(* Logix 5000 project; controller reports 1756-L63 rev 20.15; software revision 20.04; part 36 of 52 *)

        [42].log_data[40].minminute := 21, [42].log_data[40].maxminute := 25, [42].log_data[40].valid := 1, [42].log_data[41].min := 0.03412134, [42].log_data[41].max := 0.04962842, [42].log_data[41].total := 152.0447, [42].log_data[41].time := 3600.0, [42].log_data[41].minminute := 8, [42].log_data[41].maxminute := 47, [42].log_data[41].valid := 1, [42].log_data[42].min := 2.2923493, [42].log_data[42].max := 2.2970603, [42].log_data[42].total := 8261.717, [42].log_data[42].time := 3600.0, [42].log_data[42].minminute := 49, [42].log_data[42].maxminute := 24, [42].log_data[42].valid := 1, [42].log_data[43].min := -0.27999878, [42].log_data[43].max := -0.26000214, [42].log_data[43].total := -1007.5765, [42].log_data[43].time := 3600.0, [42].log_data[43].valid := 1, [42].log_data[44].min := -0.3199997, [42].log_data[44].max := -0.30000305, [42].log_data[44].total := -1084.2107, [42].log_data[44].time := 3600.0, [42].log_data[44].minminute := 1, [42].log_data[44].valid := 1, [42].log_data[45].time := 3600.0, [42].log_data[45].valid := 1, [42].log_data[46].time := 3600.0, [42].log_data[46].valid := 1, [42].log_data[47].time := 3600.0, [42].log_data[47].valid := 1, [42].log_data[48].min := 6.5827026, [42].log_data[48].max := 6.9506707, [42].log_data[48].total := 24231.43, [42].log_data[48].time := 3600.0, [42].log_data[48].minminute := 26, [42].log_data[48].maxminute := 3, [42].log_data[48].valid := 1, [42].log_data[49].min := 7.0381904, [42].log_data[49].max := 9.47083, [42].log_data[49].total := 29556.547, [42].log_data[49].time := 3600.0, [42].log_data[49].minminute := 23, [42].log_data[49].maxminute := 59, [42].log_data[49].valid := 1, [42].log_data[50].min := 2.0538552, [42].log_data[50].max := 2.1284068, [42].log_data[50].total := 7533.663, [42].log_data[50].time := 3600.0, [42].log_data[50].minminute := 59, [42].log_data[50].maxminute := 6, [42].log_data[50].valid := 1, [42].log_data[51].time := 3600.0, [42].log_data[51].valid := 1, [42].log_data[52].min := -2.959999, [42].log_data[52].max := 0.11999512, [42].log_data[52].total := -7758.8574,
        [42].log_data[52].time := 3600.0, [42].log_data[52].valid := 1, [42].log_data[53].min := -2.7400055, [42].log_data[53].max := 0.27999878, [42].log_data[53].total := -7175.7085, [42].log_data[53].time := 3600.0, [42].log_data[53].minminute := 37, [42].log_data[53].maxminute := 5, [42].log_data[53].valid := 1, [42].log_data[54].max := 0.538, [42].log_data[54].total := 1231.8954, [42].log_data[54].time := 3600.0, [42].log_data[54].maxminute := 11, [42].log_data[54].valid := 1, [42].log_data[55].max := 0.568, [42].log_data[55].total := 1217.1237, [42].log_data[55].time := 3600.0, [42].log_data[55].minminute := 4, [42].log_data[55].maxminute := 37, [42].log_data[55].valid := 1, [42].log_data[56].min := 0.16024561, [42].log_data[56].max := 0.1607167, [42].log_data[56].total := 577.47437, [42].log_data[56].time := 3600.0, [42].log_data[56].minminute := 10, [42].log_data[56].maxminute := 50, [42].log_data[56].valid := 1, [42].log_data[57].min := 0.28492987, [42].log_data[57].max := 0.28661802, [42].log_data[57].total := 1028.5197, [42].log_data[57].time := 3600.0, [42].log_data[57].minminute := 47, [42].log_data[57].maxminute := 1, [42].log_data[57].valid := 1, [42].log_data[58].time := 3600.0, [42].log_data[58].valid := 1, [42].log_data[59].time := 3600.0, [42].log_data[59].valid := 1, [42].log_data[60].valid := 1, [42].log_data[61].valid := 1, [42].log_data[62].valid := 1, [42].log_data[63].valid := 1, [42].log_data[64].valid := 1, [42].log_data[65].valid := 1, [42].log_data[66].valid := 1, [42].log_data[67].valid := 1, [42].log_data[68].valid := 1, [42].log_data[69].valid := 1, [42].log_data[70].valid := 1, [42].log_data[71].valid := 1, [42].log_data[72].valid := 1, [42].log_data[73].valid := 1, [42].log_data[74].valid := 1, [42].log_data[75].valid := 1, [42].log_data[76].valid := 1, [42].log_data[77].valid := 1, [42].log_data[78].valid := 1, [42].log_data[79].valid := 1, [42].log_data[80].valid := 1, [42].log_data[81].valid := 1,
        [42].log_data[82].valid := 1, [42].log_data[83].valid := 1, [42].log_data[84].valid := 1, [42].log_data[85].valid := 1, [42].log_data[86].valid := 1, [42].log_data[87].valid := 1, [42].log_data[88].valid := 1, [42].log_data[89].valid := 1, [42].log_data[90].valid := 1, [42].log_data[91].valid := 1, [42].log_data[92].valid := 1, [42].log_data[93].valid := 1, [42].log_data[94].valid := 1, [42].log_data[95].valid := 1, [42].log_data[96].valid := 1, [42].log_data[97].valid := 1, [42].log_data[98].valid := 1, [42].log_data[99].valid := 1, [42].log_data[100].valid := 1, [42].log_data[101].valid := 1, [42].log_data[102].valid := 1, [42].log_data[103].valid := 1, [42].log_data[104].valid := 1, [42].log_data[105].valid := 1, [42].log_data[106].valid := 1, [42].log_data[107].valid := 1, [42].log_data[108].valid := 1, [42].log_data[109].valid := 1, [42].log_data[110].valid := 1, [42].log_data[111].valid := 1, [42].log_data[112].valid := 1, [42].log_data[113].valid := 1, [42].log_data[114].valid := 1, [42].log_data[115].valid := 1, [42].log_data[116].valid := 1, [42].log_data[117].valid := 1, [42].log_data[118].valid := 1, [42].log_data[119].valid := 1, [42].log_data[120].valid := 1, [42].log_data[121].valid := 1, [42].log_data[122].valid := 1, [42].log_data[123].valid := 1, [42].log_data[124].valid := 1, [42].time.Year := 2023, [42].time.Month := 1, [42].time.Day := 14, [42].time.Hour := 21, [42].time.Minute := 59, [42].time.Second := 59, [43].log_data[0].min := 1.0, [43].log_data[0].max := 1.0, [43].log_data[0].total := 3600.0, [43].log_data[0].time := 3600.0, [43].log_data[0].valid := 1, [43].log_data[1].max := 1.0, [43].log_data[1].total := 564.5, [43].log_data[1].time := 3600.0, [43].log_data[1].maxminute := 21, [43].log_data[1].valid := 1, [43].log_data[2].max := 1.0,
        [43].log_data[2].total := 561.0, [43].log_data[2].time := 3600.0, [43].log_data[2].maxminute := 21, [43].log_data[2].valid := 1, [43].log_data[3].time := 3600.0, [43].log_data[3].valid := 1, [43].log_data[4].time := 3600.0, [43].log_data[4].valid := 1, [43].log_data[5].max := 1.0, [43].log_data[5].total := 239.5, [43].log_data[5].time := 3600.0, [43].log_data[5].maxminute := 22, [43].log_data[5].valid := 1, [43].log_data[6].time := 3600.0, [43].log_data[6].valid := 1, [43].log_data[7].time := 3600.0, [43].log_data[7].valid := 1, [43].log_data[8].min := 1.0, [43].log_data[8].max := 1.0, [43].log_data[8].total := 3600.0, [43].log_data[8].time := 3600.0, [43].log_data[8].valid := 1, [43].log_data[9].min := 1.0, [43].log_data[9].max := 1.0, [43].log_data[9].total := 3600.0, [43].log_data[9].time := 3600.0, [43].log_data[9].valid := 1, [43].log_data[10].min := 1.0, [43].log_data[10].max := 1.0, [43].log_data[10].total := 3600.0, [43].log_data[10].time := 3600.0, [43].log_data[10].valid := 1, [43].log_data[11].time := 3600.0, [43].log_data[11].valid := 1, [43].log_data[12].min := 1.0, [43].log_data[12].max := 1.0, [43].log_data[12].total := 3600.0, [43].log_data[12].time := 3600.0, [43].log_data[12].valid := 1, [43].log_data[13].min := 1.0, [43].log_data[13].max := 1.0, [43].log_data[13].total := 3600.0, [43].log_data[13].time := 3600.0, [43].log_data[13].valid := 1, [43].log_data[14].time := 3600.0, [43].log_data[14].valid := 1, [43].log_data[15].time := 3600.0, [43].log_data[15].valid := 1, [43].log_data[16].time := 3600.0, [43].log_data[16].valid := 1, [43].log_data[17].min := 1.0, [43].log_data[17].max := 1.0, [43].log_data[17].total := 3600.0, [43].log_data[17].time := 3600.0, [43].log_data[17].valid := 1, [43].log_data[18].time := 3600.0, [43].log_data[18].valid := 1, [43].log_data[19].time := 3600.0, [43].log_data[19].valid := 1, [43].log_data[20].time := 3600.0,
        [43].log_data[20].valid := 1, [43].log_data[21].min := 1.0, [43].log_data[21].max := 1.0, [43].log_data[21].total := 3600.0, [43].log_data[21].time := 3600.0, [43].log_data[21].valid := 1, [43].log_data[22].time := 3600.0, [43].log_data[22].valid := 1, [43].log_data[23].time := 3600.0, [43].log_data[23].valid := 1, [43].log_data[24].time := 3600.0, [43].log_data[24].valid := 1, [43].log_data[25].time := 3600.0, [43].log_data[25].valid := 1, [43].log_data[26].time := 3600.0, [43].log_data[26].valid := 1, [43].log_data[27].time := 3600.0, [43].log_data[27].valid := 1, [43].log_data[28].time := 3600.0, [43].log_data[28].valid := 1, [43].log_data[29].min := 1.0, [43].log_data[29].max := 1.0, [43].log_data[29].total := 3600.0, [43].log_data[29].time := 3600.0, [43].log_data[29].valid := 1, [43].log_data[30].min := 1.0, [43].log_data[30].max := 1.0, [43].log_data[30].total := 3600.0, [43].log_data[30].time := 3600.0, [43].log_data[30].valid := 1, [43].log_data[31].max := 1.0, [43].log_data[31].total := 1629.998, [43].log_data[31].time := 3600.0, [43].log_data[31].maxminute := 3, [43].log_data[31].valid := 1, [43].log_data[32].max := 1.0, [43].log_data[32].total := 1440.998, [43].log_data[32].time := 3600.0, [43].log_data[32].minminute := 2, [43].log_data[32].valid := 1, [43].log_data[33].time := 3600.0, [43].log_data[33].valid := 1, [43].log_data[34].time := 3600.0, [43].log_data[34].valid := 1, [43].log_data[35].max := 1.0, [43].log_data[35].total := 1536.498, [43].log_data[35].time := 3600.0, [43].log_data[35].minminute := 7, [43].log_data[35].valid := 1, [43].log_data[36].max := 1.0, [43].log_data[36].total := 1622.2471, [43].log_data[36].time := 3600.0, [43].log_data[36].maxminute := 8, [43].log_data[36].valid := 1, [43].log_data[37].max := 7.23916, [43].log_data[37].total := 3552.5513, [43].log_data[37].time := 3600.0, [43].log_data[37].maxminute := 23, [43].log_data[37].valid := 1, [43].log_data[38].time := 3600.0,
        [43].log_data[38].valid := 1, [43].log_data[39].min := 0.997415, [43].log_data[39].max := 1.0214411, [43].log_data[39].total := 3638.9631, [43].log_data[39].time := 3600.0, [43].log_data[39].minminute := 29, [43].log_data[39].maxminute := 26, [43].log_data[39].valid := 1, [43].log_data[40].min := 7.5816298, [43].log_data[40].max := 7.5865765, [43].log_data[40].total := 27307.055, [43].log_data[40].time := 3600.0, [43].log_data[40].minminute := 41, [43].log_data[40].maxminute := 2, [43].log_data[40].valid := 1, [43].log_data[41].min := 0.03785083, [43].log_data[41].max := 0.056694824, [43].log_data[41].total := 165.39845, [43].log_data[41].time := 3600.0, [43].log_data[41].minminute := 46, [43].log_data[41].maxminute := 20, [43].log_data[41].valid := 1, [43].log_data[42].min := 2.2922316, [43].log_data[42].max := 2.2970603, [43].log_data[42].total := 8261.55, [43].log_data[42].time := 3600.0, [43].log_data[42].minminute := 23, [43].log_data[42].maxminute := 1, [43].log_data[42].valid := 1, [43].log_data[43].min := -0.27999878, [43].log_data[43].max := -0.26000214, [43].log_data[43].total := -1007.7663, [43].log_data[43].time := 3600.0, [43].log_data[43].maxminute := 10, [43].log_data[43].valid := 1, [43].log_data[44].min := -0.3199997, [43].log_data[44].max := -0.30000305, [43].log_data[44].total := -1084.6222, [43].log_data[44].time := 3600.0, [43].log_data[44].valid := 1, [43].log_data[45].time := 3600.0, [43].log_data[45].valid := 1, [43].log_data[46].time := 3600.0, [43].log_data[46].valid := 1, [43].log_data[47].time := 3600.0, [43].log_data[47].valid := 1, [43].log_data[48].min := 6.5794053, [43].log_data[48].max := 6.9666095, [43].log_data[48].total := 24206.664, [43].log_data[48].time := 3600.0, [43].log_data[48].minminute := 53, [43].log_data[48].maxminute := 29, [43].log_data[48].valid := 1, [43].log_data[49].min := 6.964974, [43].log_data[49].max := 9.644745, [43].log_data[49].total := 30286.188, [43].log_data[49].time := 3600.0, [43].log_data[49].minminute := 49, [43].log_data[49].maxminute := 20, [43].log_data[49].valid := 1,
        [43].log_data[50].min := 2.0134585, [43].log_data[50].max := 2.1326468, [43].log_data[50].total := 7487.468, [43].log_data[50].time := 3600.0, [43].log_data[50].minminute := 22, [43].log_data[50].maxminute := 30, [43].log_data[50].valid := 1, [43].log_data[51].time := 3600.0, [43].log_data[51].valid := 1, [43].log_data[52].min := -2.959999, [43].log_data[52].max := 0.11999512, [43].log_data[52].total := -7728.6436, [43].log_data[52].time := 3600.0, [43].log_data[52].minminute := 4, [43].log_data[52].maxminute := 2, [43].log_data[52].valid := 1, [43].log_data[53].min := -2.5200043, [43].log_data[53].max := 0.27999878, [43].log_data[53].total := -7386.8955, [43].log_data[53].time := 3600.0, [43].log_data[53].minminute := 55, [43].log_data[53].maxminute := 51, [43].log_data[53].valid := 1, [43].log_data[54].max := 0.523, [43].log_data[54].total := 1217.3251, [43].log_data[54].time := 3600.0, [43].log_data[54].minminute := 2, [43].log_data[54].maxminute := 25, [43].log_data[54].valid := 1, [43].log_data[55].max := 0.522, [43].log_data[55].total := 1254.3055, [43].log_data[55].time := 3600.0, [43].log_data[55].minminute := 7, [43].log_data[55].maxminute := 40, [43].log_data[55].valid := 1, [43].log_data[56].min := 0.16020635, [43].log_data[56].max := 0.16067745, [43].log_data[56].total := 577.47656, [43].log_data[56].time := 3600.0, [43].log_data[56].minminute := 57, [43].log_data[56].maxminute := 11, [43].log_data[56].valid := 1, [43].log_data[57].min := 0.28355587, [43].log_data[57].max := 0.28532246, [43].log_data[57].total := 1025.724, [43].log_data[57].time := 3600.0, [43].log_data[57].minminute := 59, [43].log_data[57].maxminute := 11, [43].log_data[57].valid := 1, [43].log_data[58].time := 3600.0, [43].log_data[58].valid := 1, [43].log_data[59].time := 3600.0, [43].log_data[59].valid := 1, [43].log_data[60].valid := 1, [43].log_data[61].valid := 1, [43].log_data[62].valid := 1, [43].log_data[63].valid := 1, [43].log_data[64].valid := 1, [43].log_data[65].valid := 1, [43].log_data[66].valid := 1,
        [43].log_data[67].valid := 1, [43].log_data[68].valid := 1, [43].log_data[69].valid := 1, [43].log_data[70].valid := 1, [43].log_data[71].valid := 1, [43].log_data[72].valid := 1, [43].log_data[73].valid := 1, [43].log_data[74].valid := 1, [43].log_data[75].valid := 1, [43].log_data[76].valid := 1, [43].log_data[77].valid := 1, [43].log_data[78].valid := 1, [43].log_data[79].valid := 1, [43].log_data[80].valid := 1, [43].log_data[81].valid := 1, [43].log_data[82].valid := 1, [43].log_data[83].valid := 1, [43].log_data[84].valid := 1, [43].log_data[85].valid := 1, [43].log_data[86].valid := 1, [43].log_data[87].valid := 1, [43].log_data[88].valid := 1, [43].log_data[89].valid := 1, [43].log_data[90].valid := 1, [43].log_data[91].valid := 1, [43].log_data[92].valid := 1, [43].log_data[93].valid := 1, [43].log_data[94].valid := 1, [43].log_data[95].valid := 1, [43].log_data[96].valid := 1, [43].log_data[97].valid := 1, [43].log_data[98].valid := 1, [43].log_data[99].valid := 1, [43].log_data[100].valid := 1, [43].log_data[101].valid := 1, [43].log_data[102].valid := 1, [43].log_data[103].valid := 1, [43].log_data[104].valid := 1, [43].log_data[105].valid := 1, [43].log_data[106].valid := 1, [43].log_data[107].valid := 1, [43].log_data[108].valid := 1, [43].log_data[109].valid := 1, [43].log_data[110].valid := 1, [43].log_data[111].valid := 1, [43].log_data[112].valid := 1, [43].log_data[113].valid := 1, [43].log_data[114].valid := 1, [43].log_data[115].valid := 1, [43].log_data[116].valid := 1, [43].log_data[117].valid := 1, [43].log_data[118].valid := 1, [43].log_data[119].valid := 1, [43].log_data[120].valid := 1, [43].log_data[121].valid := 1, [43].log_data[122].valid := 1, [43].log_data[123].valid := 1, [43].log_data[124].valid := 1, [43].time.Year := 2023, [43].time.Month := 1,
        [43].time.Day := 14, [43].time.Hour := 22, [43].time.Minute := 59, [43].time.Second := 59, [44].log_data[0].min := 1.0, [44].log_data[0].max := 1.0, [44].log_data[0].total := 3599.5, [44].log_data[0].time := 3599.5, [44].log_data[0].valid := 1, [44].log_data[1].max := 1.0, [44].log_data[1].total := 535.5, [44].log_data[1].time := 3599.5, [44].log_data[1].maxminute := 50, [44].log_data[1].valid := 1, [44].log_data[2].max := 1.0, [44].log_data[2].total := 532.0, [44].log_data[2].time := 3599.5, [44].log_data[2].maxminute := 50, [44].log_data[2].valid := 1, [44].log_data[3].time := 3599.5, [44].log_data[3].valid := 1, [44].log_data[4].time := 3599.5, [44].log_data[4].valid := 1, [44].log_data[5].max := 1.0, [44].log_data[5].total := 227.5, [44].log_data[5].time := 3599.5, [44].log_data[5].maxminute := 51, [44].log_data[5].valid := 1, [44].log_data[6].time := 3599.5, [44].log_data[6].valid := 1, [44].log_data[7].time := 3599.5, [44].log_data[7].valid := 1, [44].log_data[8].min := 1.0, [44].log_data[8].max := 1.0, [44].log_data[8].total := 3599.5, [44].log_data[8].time := 3599.5, [44].log_data[8].valid := 1, [44].log_data[9].min := 1.0, [44].log_data[9].max := 1.0, [44].log_data[9].total := 3599.5, [44].log_data[9].time := 3599.5, [44].log_data[9].valid := 1, [44].log_data[10].min := 1.0, [44].log_data[10].max := 1.0, [44].log_data[10].total := 3599.5, [44].log_data[10].time := 3599.5, [44].log_data[10].valid := 1, [44].log_data[11].time := 3599.5, [44].log_data[11].valid := 1, [44].log_data[12].min := 1.0, [44].log_data[12].max := 1.0, [44].log_data[12].total := 3599.5, [44].log_data[12].time := 3599.5, [44].log_data[12].valid := 1, [44].log_data[13].min := 1.0, [44].log_data[13].max := 1.0, [44].log_data[13].total := 3599.5, [44].log_data[13].time := 3599.5, [44].log_data[13].valid := 1, [44].log_data[14].time := 3599.5,
        [44].log_data[14].valid := 1, [44].log_data[15].time := 3599.5, [44].log_data[15].valid := 1, [44].log_data[16].time := 3599.5, [44].log_data[16].valid := 1, [44].log_data[17].min := 1.0, [44].log_data[17].max := 1.0, [44].log_data[17].total := 3599.5, [44].log_data[17].time := 3599.5, [44].log_data[17].valid := 1, [44].log_data[18].time := 3599.5, [44].log_data[18].valid := 1, [44].log_data[19].time := 3599.5, [44].log_data[19].valid := 1, [44].log_data[20].time := 3599.5, [44].log_data[20].valid := 1, [44].log_data[21].min := 1.0, [44].log_data[21].max := 1.0, [44].log_data[21].total := 3599.5, [44].log_data[21].time := 3599.5, [44].log_data[21].valid := 1, [44].log_data[22].time := 3599.5, [44].log_data[22].valid := 1, [44].log_data[23].time := 3599.5, [44].log_data[23].valid := 1, [44].log_data[24].time := 3599.5, [44].log_data[24].valid := 1, [44].log_data[25].time := 3599.5, [44].log_data[25].valid := 1, [44].log_data[26].time := 3599.5, [44].log_data[26].valid := 1, [44].log_data[27].time := 3599.5, [44].log_data[27].valid := 1, [44].log_data[28].time := 3599.5, [44].log_data[28].valid := 1, [44].log_data[29].min := 1.0, [44].log_data[29].max := 1.0, [44].log_data[29].total := 3599.5, [44].log_data[29].time := 3599.5, [44].log_data[29].valid := 1, [44].log_data[30].min := 1.0, [44].log_data[30].max := 1.0, [44].log_data[30].total := 3599.5, [44].log_data[30].time := 3599.5, [44].log_data[30].valid := 1, [44].log_data[31].max := 1.0, [44].log_data[31].total := 1629.7471, [44].log_data[31].time := 3599.5, [44].log_data[31].maxminute := 7, [44].log_data[31].valid := 1, [44].log_data[32].max := 1.0, [44].log_data[32].total := 1440.498, [44].log_data[32].time := 3599.5, [44].log_data[32].minminute := 5, [44].log_data[32].valid := 1, [44].log_data[33].time := 3599.5, [44].log_data[33].valid := 1, [44].log_data[34].time := 3599.5, [44].log_data[34].valid := 1, [44].log_data[35].max := 1.0,
        [44].log_data[35].total := 1629.7471, [44].log_data[35].time := 3599.5, [44].log_data[35].maxminute := 1, [44].log_data[35].valid := 1, [44].log_data[36].max := 1.0, [44].log_data[36].total := 1440.2471, [44].log_data[36].time := 3599.5, [44].log_data[36].valid := 1, [44].log_data[37].max := 7.5873804, [44].log_data[37].total := 3523.6545, [44].log_data[37].time := 3599.5, [44].log_data[37].maxminute := 52, [44].log_data[37].valid := 1, [44].log_data[38].time := 3599.5, [44].log_data[38].valid := 1, [44].log_data[39].min := 0.99859273, [44].log_data[39].max := 1.0223833, [44].log_data[39].total := 3639.1343, [44].log_data[39].time := 3599.5, [44].log_data[39].minminute := 53, [44].log_data[39].maxminute := 51, [44].log_data[39].valid := 1, [44].log_data[40].min := 7.5703626, [44].log_data[40].max := 7.592072, [44].log_data[40].total := 27304.006, [44].log_data[40].time := 3599.5, [44].log_data[40].minminute := 57, [44].log_data[40].maxminute := 58, [44].log_data[40].valid := 1, [44].log_data[41].min := 0.029802978, [44].log_data[41].max := 0.044524662, [44].log_data[41].total := 127.272896, [44].log_data[41].time := 3599.5, [44].log_data[41].minminute := 15, [44].log_data[41].valid := 1, [44].log_data[42].min := 2.2921138, [44].log_data[42].max := 2.2970603, [44].log_data[42].total := 8260.388, [44].log_data[42].time := 3599.5, [44].log_data[42].minminute := 50, [44].log_data[42].maxminute := 11, [44].log_data[42].valid := 1, [44].log_data[43].min := -0.27999878, [44].log_data[43].max := -0.26000214, [44].log_data[43].total := -1004.873, [44].log_data[43].time := 3599.5, [44].log_data[43].valid := 1, [44].log_data[44].min := -0.3199997, [44].log_data[44].max := -0.30000305, [44].log_data[44].total := -1081.1991, [44].log_data[44].time := 3599.5, [44].log_data[44].valid := 1, [44].log_data[45].time := 3599.5, [44].log_data[45].valid := 1, [44].log_data[46].time := 3599.5, [44].log_data[46].valid := 1, [44].log_data[47].time := 3599.5, [44].log_data[47].valid := 1, [44].log_data[48].min := 6.690153, [44].log_data[48].max := 6.9295106,
        [44].log_data[48].total := 24392.291, [44].log_data[48].time := 3599.5, [44].log_data[48].maxminute := 57, [44].log_data[48].valid := 1, [44].log_data[49].min := 7.833956, [44].log_data[49].max := 9.64494, [44].log_data[49].total := 33088.74, [44].log_data[49].time := 3599.5, [44].log_data[49].maxminute := 50, [44].log_data[49].valid := 1, [44].log_data[50].min := 2.006392, [44].log_data[50].max := 2.1253445, [44].log_data[50].total := 7408.252, [44].log_data[50].time := 3599.5, [44].log_data[50].minminute := 51, [44].log_data[50].maxminute := 57, [44].log_data[50].valid := 1, [44].log_data[51].time := 3599.5, [44].log_data[51].valid := 1, [44].log_data[52].min := -3.0999985, [44].log_data[52].max := 0.11999512, [44].log_data[52].total := -7716.6855, [44].log_data[52].time := 3599.5, [44].log_data[52].minminute := 7, [44].log_data[52].maxminute := 5, [44].log_data[52].valid := 1, [44].log_data[53].min := -2.5, [44].log_data[53].max := 0.27999878, [44].log_data[53].total := -7181.388, [44].log_data[53].time := 3599.5, [44].log_data[53].minminute := 4, [44].log_data[53].maxminute := 43, [44].log_data[53].valid := 1, [44].log_data[54].max := 0.55149996, [44].log_data[54].total := 1217.8906, [44].log_data[54].time := 3599.5, [44].log_data[54].minminute := 5, [44].log_data[54].maxminute := 49, [44].log_data[54].valid := 1, [44].log_data[55].max := 0.5395, [44].log_data[55].total := 1217.0914, [44].log_data[55].time := 3599.5, [44].log_data[55].maxminute := 22, [44].log_data[55].valid := 1, [44].log_data[56].min := 0.16028486, [44].log_data[56].max := 0.16063818, [44].log_data[56].total := 577.4504, [44].log_data[56].time := 3599.5, [44].log_data[56].minminute := 14, [44].log_data[56].maxminute := 3, [44].log_data[56].valid := 1, [44].log_data[57].min := 0.2833203, [44].log_data[57].max := 0.2837129, [44].log_data[57].total := 1020.4592, [44].log_data[57].time := 3599.5, [44].log_data[57].minminute := 32, [44].log_data[57].valid := 1, [44].log_data[58].time := 3599.5, [44].log_data[58].valid := 1, [44].log_data[59].time := 3599.5,
        [44].log_data[59].valid := 1, [44].log_data[60].valid := 1, [44].log_data[61].valid := 1, [44].log_data[62].valid := 1, [44].log_data[63].valid := 1, [44].log_data[64].valid := 1, [44].log_data[65].valid := 1, [44].log_data[66].valid := 1, [44].log_data[67].valid := 1, [44].log_data[68].valid := 1, [44].log_data[69].valid := 1, [44].log_data[70].valid := 1, [44].log_data[71].valid := 1, [44].log_data[72].valid := 1, [44].log_data[73].valid := 1, [44].log_data[74].valid := 1, [44].log_data[75].valid := 1, [44].log_data[76].valid := 1, [44].log_data[77].valid := 1, [44].log_data[78].valid := 1, [44].log_data[79].valid := 1, [44].log_data[80].valid := 1, [44].log_data[81].valid := 1, [44].log_data[82].valid := 1, [44].log_data[83].valid := 1, [44].log_data[84].valid := 1, [44].log_data[85].valid := 1, [44].log_data[86].valid := 1, [44].log_data[87].valid := 1, [44].log_data[88].valid := 1, [44].log_data[89].valid := 1, [44].log_data[90].valid := 1, [44].log_data[91].valid := 1, [44].log_data[92].valid := 1, [44].log_data[93].valid := 1, [44].log_data[94].valid := 1, [44].log_data[95].valid := 1, [44].log_data[96].valid := 1, [44].log_data[97].valid := 1, [44].log_data[98].valid := 1, [44].log_data[99].valid := 1, [44].log_data[100].valid := 1, [44].log_data[101].valid := 1, [44].log_data[102].valid := 1, [44].log_data[103].valid := 1, [44].log_data[104].valid := 1, [44].log_data[105].valid := 1, [44].log_data[106].valid := 1, [44].log_data[107].valid := 1, [44].log_data[108].valid := 1, [44].log_data[109].valid := 1, [44].log_data[110].valid := 1, [44].log_data[111].valid := 1, [44].log_data[112].valid := 1, [44].log_data[113].valid := 1, [44].log_data[114].valid := 1, [44].log_data[115].valid := 1, [44].log_data[116].valid := 1, [44].log_data[117].valid := 1, [44].log_data[118].valid := 1,
        [44].log_data[119].valid := 1, [44].log_data[120].valid := 1, [44].log_data[121].valid := 1, [44].log_data[122].valid := 1, [44].log_data[123].valid := 1, [44].log_data[124].valid := 1, [44].time.Year := 2023, [44].time.Month := 1, [44].time.Day := 14, [44].time.Hour := 23, [44].time.Minute := 59, [44].time.Second := 59, [45].log_data[0].min := 1.0, [45].log_data[0].max := 1.0, [45].log_data[0].total := 3600.0, [45].log_data[0].time := 3600.0, [45].log_data[0].valid := 1, [45].log_data[1].time := 3600.0, [45].log_data[1].valid := 1, [45].log_data[2].time := 3600.0, [45].log_data[2].valid := 1, [45].log_data[3].time := 3600.0, [45].log_data[3].valid := 1, [45].log_data[4].time := 3600.0, [45].log_data[4].valid := 1, [45].log_data[5].time := 3600.0, [45].log_data[5].valid := 1, [45].log_data[6].time := 3600.0, [45].log_data[6].valid := 1, [45].log_data[7].time := 3600.0, [45].log_data[7].valid := 1, [45].log_data[8].min := 1.0, [45].log_data[8].max := 1.0, [45].log_data[8].total := 3600.0, [45].log_data[8].time := 3600.0, [45].log_data[8].valid := 1, [45].log_data[9].min := 1.0, [45].log_data[9].max := 1.0, [45].log_data[9].total := 3600.0, [45].log_data[9].time := 3600.0, [45].log_data[9].valid := 1, [45].log_data[10].min := 1.0, [45].log_data[10].max := 1.0, [45].log_data[10].total := 3600.0, [45].log_data[10].time := 3600.0, [45].log_data[10].valid := 1, [45].log_data[11].time := 3600.0, [45].log_data[11].valid := 1, [45].log_data[12].min := 1.0, [45].log_data[12].max := 1.0, [45].log_data[12].total := 3600.0, [45].log_data[12].time := 3600.0, [45].log_data[12].valid := 1, [45].log_data[13].min := 1.0, [45].log_data[13].max := 1.0, [45].log_data[13].total := 3600.0, [45].log_data[13].time := 3600.0, [45].log_data[13].valid := 1, [45].log_data[14].time := 3600.0, [45].log_data[14].valid := 1,
        [45].log_data[15].time := 3600.0, [45].log_data[15].valid := 1, [45].log_data[16].time := 3600.0, [45].log_data[16].valid := 1, [45].log_data[17].min := 1.0, [45].log_data[17].max := 1.0, [45].log_data[17].total := 3600.0, [45].log_data[17].time := 3600.0, [45].log_data[17].valid := 1, [45].log_data[18].time := 3600.0, [45].log_data[18].valid := 1, [45].log_data[19].time := 3600.0, [45].log_data[19].valid := 1, [45].log_data[20].time := 3600.0, [45].log_data[20].valid := 1, [45].log_data[21].min := 1.0, [45].log_data[21].max := 1.0, [45].log_data[21].total := 3600.0, [45].log_data[21].time := 3600.0, [45].log_data[21].valid := 1, [45].log_data[22].time := 3600.0, [45].log_data[22].valid := 1, [45].log_data[23].time := 3600.0, [45].log_data[23].valid := 1, [45].log_data[24].time := 3600.0, [45].log_data[24].valid := 1, [45].log_data[25].time := 3600.0, [45].log_data[25].valid := 1, [45].log_data[26].time := 3600.0, [45].log_data[26].valid := 1, [45].log_data[27].time := 3600.0, [45].log_data[27].valid := 1, [45].log_data[28].time := 3600.0, [45].log_data[28].valid := 1, [45].log_data[29].min := 1.0, [45].log_data[29].max := 1.0, [45].log_data[29].total := 3600.0, [45].log_data[29].time := 3600.0, [45].log_data[29].valid := 1, [45].log_data[30].min := 1.0, [45].log_data[30].max := 1.0, [45].log_data[30].total := 3600.0, [45].log_data[30].time := 3600.0, [45].log_data[30].valid := 1, [45].log_data[31].max := 1.0, [45].log_data[31].total := 1542.2471, [45].log_data[31].time := 3600.0, [45].log_data[31].maxminute := 10, [45].log_data[31].valid := 1, [45].log_data[32].max := 1.0, [45].log_data[32].total := 1616.498, [45].log_data[32].time := 3600.0, [45].log_data[32].minminute := 8, [45].log_data[32].valid := 1, [45].log_data[33].time := 3600.0, [45].log_data[33].valid := 1, [45].log_data[34].time := 3600.0, [45].log_data[34].valid := 1, [45].log_data[35].max := 1.0, [45].log_data[35].total := 1629.998,
        [45].log_data[35].time := 3600.0, [45].log_data[35].maxminute := 4, [45].log_data[35].valid := 1, [45].log_data[36].max := 1.0, [45].log_data[36].total := 1440.7471, [45].log_data[36].time := 3600.0, [45].log_data[36].minminute := 3, [45].log_data[36].valid := 1, [45].log_data[37].time := 3600.0, [45].log_data[37].valid := 1, [45].log_data[38].time := 3600.0, [45].log_data[38].valid := 1, [45].log_data[39].min := 1.0050704, [45].log_data[39].max := 1.0186145, [45].log_data[39].total := 3648.3677, [45].log_data[39].time := 3600.0, [45].log_data[39].minminute := 13, [45].log_data[39].maxminute := 55, [45].log_data[39].valid := 1, [45].log_data[40].min := 7.561569, [45].log_data[40].max := 7.5934467, [45].log_data[40].total := 27307.957, [45].log_data[40].time := 3600.0, [45].log_data[40].minminute := 18, [45].log_data[40].maxminute := 20, [45].log_data[40].valid := 1, [45].log_data[41].min := 0.030980714, [45].log_data[41].max := 0.052572753, [45].log_data[41].total := 154.78441, [45].log_data[41].time := 3600.0, [45].log_data[41].minminute := 11, [45].log_data[41].maxminute := 47, [45].log_data[41].valid := 1, [45].log_data[42].min := 2.292467, [45].log_data[42].max := 2.2968247, [45].log_data[42].total := 8261.483, [45].log_data[42].time := 3600.0, [45].log_data[42].minminute := 9, [45].log_data[42].maxminute := 12, [45].log_data[42].valid := 1, [45].log_data[43].min := -0.27999878, [45].log_data[43].max := -0.26000214, [45].log_data[43].total := -1006.5029, [45].log_data[43].time := 3600.0, [45].log_data[43].valid := 1, [45].log_data[44].min := -0.3199997, [45].log_data[44].max := -0.30000305, [45].log_data[44].total := -1080.491, [45].log_data[44].time := 3600.0, [45].log_data[44].minminute := 2, [45].log_data[44].valid := 1, [45].log_data[45].time := 3600.0, [45].log_data[45].valid := 1, [45].log_data[46].time := 3600.0, [45].log_data[46].valid := 1, [45].log_data[47].time := 3600.0, [45].log_data[47].valid := 1, [45].log_data[48].min := 6.5810537, [45].log_data[48].max := 6.819587, [45].log_data[48].total := 24196.793,
        [45].log_data[48].time := 3600.0, [45].log_data[48].minminute := 21, [45].log_data[48].valid := 1, [45].log_data[49].min := 6.9233603, [45].log_data[49].max := 9.528736, [45].log_data[49].total := 29744.072, [45].log_data[49].time := 3600.0, [45].log_data[49].minminute := 17, [45].log_data[49].maxminute := 59, [45].log_data[49].valid := 1, [45].log_data[50].min := 2.0334802, [45].log_data[50].max := 2.120398, [45].log_data[50].total := 7473.879, [45].log_data[50].time := 3600.0, [45].log_data[50].minminute := 59, [45].log_data[50].maxminute := 1, [45].log_data[50].valid := 1, [45].log_data[51].time := 3600.0, [45].log_data[51].valid := 1, [45].log_data[52].min := -3.0200043, [45].log_data[52].max := 0.11999512, [45].log_data[52].total := -7984.632, [45].log_data[52].time := 3600.0, [45].log_data[52].minminute := 52, [45].log_data[52].maxminute := 9, [45].log_data[52].valid := 1, [45].log_data[53].min := -2.5200043, [45].log_data[53].max := 0.2599945, [45].log_data[53].total := -7218.632, [45].log_data[53].time := 3600.0, [45].log_data[53].minminute := 48, [45].log_data[53].maxminute := 14, [45].log_data[53].valid := 1, [45].log_data[54].max := 0.5275, [45].log_data[54].total := 1253.7211, [45].log_data[54].time := 3600.0, [45].log_data[54].minminute := 8, [45].log_data[54].maxminute := 52, [45].log_data[54].valid := 1, [45].log_data[55].max := 0.536, [45].log_data[55].total := 1217.2065, [45].log_data[55].time := 3600.0, [45].log_data[55].minminute := 3, [45].log_data[55].maxminute := 4, [45].log_data[55].valid := 1, [45].log_data[56].min := 0.16020635, [45].log_data[56].max := 0.16063818, [45].log_data[56].total := 577.4949, [45].log_data[56].time := 3600.0, [45].log_data[56].minminute := 22, [45].log_data[56].maxminute := 11, [45].log_data[56].valid := 1, [45].log_data[57].min := 0.2814752, [45].log_data[57].max := 0.28375214, [45].log_data[57].total := 1016.5351, [45].log_data[57].time := 3600.0, [45].log_data[57].minminute := 43, [45].log_data[57].maxminute := 1, [45].log_data[57].valid := 1, [45].log_data[58].time := 3600.0,
        [45].log_data[58].valid := 1, [45].log_data[59].time := 3600.0, [45].log_data[59].valid := 1, [45].log_data[60].valid := 1, [45].log_data[61].valid := 1, [45].log_data[62].valid := 1, [45].log_data[63].valid := 1, [45].log_data[64].valid := 1, [45].log_data[65].valid := 1, [45].log_data[66].valid := 1, [45].log_data[67].valid := 1, [45].log_data[68].valid := 1, [45].log_data[69].valid := 1, [45].log_data[70].valid := 1, [45].log_data[71].valid := 1, [45].log_data[72].valid := 1, [45].log_data[73].valid := 1, [45].log_data[74].valid := 1, [45].log_data[75].valid := 1, [45].log_data[76].valid := 1, [45].log_data[77].valid := 1, [45].log_data[78].valid := 1, [45].log_data[79].valid := 1, [45].log_data[80].valid := 1, [45].log_data[81].valid := 1, [45].log_data[82].valid := 1, [45].log_data[83].valid := 1, [45].log_data[84].valid := 1, [45].log_data[85].valid := 1, [45].log_data[86].valid := 1, [45].log_data[87].valid := 1, [45].log_data[88].valid := 1, [45].log_data[89].valid := 1, [45].log_data[90].valid := 1, [45].log_data[91].valid := 1, [45].log_data[92].valid := 1, [45].log_data[93].valid := 1, [45].log_data[94].valid := 1, [45].log_data[95].valid := 1, [45].log_data[96].valid := 1, [45].log_data[97].valid := 1, [45].log_data[98].valid := 1, [45].log_data[99].valid := 1, [45].log_data[100].valid := 1, [45].log_data[101].valid := 1, [45].log_data[102].valid := 1, [45].log_data[103].valid := 1, [45].log_data[104].valid := 1, [45].log_data[105].valid := 1, [45].log_data[106].valid := 1, [45].log_data[107].valid := 1, [45].log_data[108].valid := 1, [45].log_data[109].valid := 1, [45].log_data[110].valid := 1, [45].log_data[111].valid := 1, [45].log_data[112].valid := 1, [45].log_data[113].valid := 1, [45].log_data[114].valid := 1, [45].log_data[115].valid := 1, [45].log_data[116].valid := 1,
        [45].log_data[117].valid := 1, [45].log_data[118].valid := 1, [45].log_data[119].valid := 1, [45].log_data[120].valid := 1, [45].log_data[121].valid := 1, [45].log_data[122].valid := 1, [45].log_data[123].valid := 1, [45].log_data[124].valid := 1, [45].time.Year := 2023, [45].time.Month := 1, [45].time.Day := 15, [45].time.Minute := 59, [45].time.Second := 59, [46].log_data[0].min := 1.0, [46].log_data[0].max := 1.0, [46].log_data[0].total := 3600.0, [46].log_data[0].time := 3600.0, [46].log_data[0].valid := 1, [46].log_data[1].max := 1.0, [46].log_data[1].total := 550.0, [46].log_data[1].time := 3600.0, [46].log_data[1].maxminute := 40, [46].log_data[1].valid := 1, [46].log_data[2].max := 1.0, [46].log_data[2].total := 546.5, [46].log_data[2].time := 3600.0, [46].log_data[2].maxminute := 40, [46].log_data[2].valid := 1, [46].log_data[3].time := 3600.0, [46].log_data[3].valid := 1, [46].log_data[4].time := 3600.0, [46].log_data[4].valid := 1, [46].log_data[5].max := 1.0, [46].log_data[5].total := 240.0, [46].log_data[5].time := 3600.0, [46].log_data[5].maxminute := 41, [46].log_data[5].valid := 1, [46].log_data[6].time := 3600.0, [46].log_data[6].valid := 1, [46].log_data[7].time := 3600.0, [46].log_data[7].valid := 1, [46].log_data[8].max := 1.0, [46].log_data[8].total := 2416.5, [46].log_data[8].time := 3600.0, [46].log_data[8].minminute := 23, [46].log_data[8].valid := 1, [46].log_data[9].max := 1.0, [46].log_data[9].total := 2413.0, [46].log_data[9].time := 3600.0, [46].log_data[9].minminute := 23, [46].log_data[9].valid := 1, [46].log_data[10].min := 1.0, [46].log_data[10].max := 1.0, [46].log_data[10].total := 3600.0, [46].log_data[10].time := 3600.0, [46].log_data[10].valid := 1, [46].log_data[11].time := 3600.0, [46].log_data[11].valid := 1, [46].log_data[12].min := 1.0, [46].log_data[12].max := 1.0,
        [46].log_data[12].total := 3600.0, [46].log_data[12].time := 3600.0, [46].log_data[12].valid := 1, [46].log_data[13].min := 1.0, [46].log_data[13].max := 1.0, [46].log_data[13].total := 3600.0, [46].log_data[13].time := 3600.0, [46].log_data[13].valid := 1, [46].log_data[14].time := 3600.0, [46].log_data[14].valid := 1, [46].log_data[15].time := 3600.0, [46].log_data[15].valid := 1, [46].log_data[16].time := 3600.0, [46].log_data[16].valid := 1, [46].log_data[17].min := 1.0, [46].log_data[17].max := 1.0, [46].log_data[17].total := 3600.0, [46].log_data[17].time := 3600.0, [46].log_data[17].valid := 1, [46].log_data[18].time := 3600.0, [46].log_data[18].valid := 1, [46].log_data[19].time := 3600.0, [46].log_data[19].valid := 1, [46].log_data[20].time := 3600.0, [46].log_data[20].valid := 1, [46].log_data[21].min := 1.0, [46].log_data[21].max := 1.0, [46].log_data[21].total := 3600.0, [46].log_data[21].time := 3600.0, [46].log_data[21].valid := 1, [46].log_data[22].time := 3600.0, [46].log_data[22].valid := 1, [46].log_data[23].time := 3600.0, [46].log_data[23].valid := 1, [46].log_data[24].time := 3600.0, [46].log_data[24].valid := 1, [46].log_data[25].time := 3600.0, [46].log_data[25].valid := 1, [46].log_data[26].time := 3600.0, [46].log_data[26].valid := 1, [46].log_data[27].time := 3600.0, [46].log_data[27].valid := 1, [46].log_data[28].time := 3600.0, [46].log_data[28].valid := 1, [46].log_data[29].min := 1.0, [46].log_data[29].max := 1.0, [46].log_data[29].total := 3600.0, [46].log_data[29].time := 3600.0, [46].log_data[29].valid := 1, [46].log_data[30].min := 1.0, [46].log_data[30].max := 1.0, [46].log_data[30].total := 3600.0, [46].log_data[30].time := 3600.0, [46].log_data[30].valid := 1, [46].log_data[31].max := 1.0, [46].log_data[31].total := 1018.99805, [46].log_data[31].time := 3600.0, [46].log_data[31].minminute := 1, [46].log_data[31].valid := 1, [46].log_data[32].max := 1.0,
        [46].log_data[32].total := 1086.498, [46].log_data[32].time := 3600.0, [46].log_data[32].maxminute := 2, [46].log_data[32].valid := 1, [46].log_data[33].time := 3600.0, [46].log_data[33].valid := 1, [46].log_data[34].time := 3600.0, [46].log_data[34].valid := 1, [46].log_data[35].max := 1.0, [46].log_data[35].total := 839.7471, [46].log_data[35].time := 3600.0, [46].log_data[35].maxminute := 7, [46].log_data[35].valid := 1, [46].log_data[36].max := 1.0, [46].log_data[36].total := 1216.998, [46].log_data[36].time := 3600.0, [46].log_data[36].minminute := 6, [46].log_data[36].valid := 1, [46].log_data[37].max := 7.2364116, [46].log_data[37].total := 3456.245, [46].log_data[37].time := 3600.0, [46].log_data[37].maxminute := 41, [46].log_data[37].valid := 1, [46].log_data[38].time := 3600.0, [46].log_data[38].valid := 1, [46].log_data[39].min := 0.9971795, [46].log_data[39].max := 1.0216767, [46].log_data[39].total := 3645.0046, [46].log_data[39].time := 3600.0, [46].log_data[39].minminute := 43, [46].log_data[39].maxminute := 41, [46].log_data[39].valid := 1, [46].log_data[40].min := 7.561844, [46].log_data[40].max := 7.597843, [46].log_data[40].total := 27306.037, [46].log_data[40].time := 3600.0, [46].log_data[40].minminute := 26, [46].log_data[40].maxminute := 33, [46].log_data[40].valid := 1, [46].log_data[41].min := 0.03588794, [46].log_data[41].max := 0.058657713, [46].log_data[41].total := 164.50613, [46].log_data[41].time := 3600.0, [46].log_data[41].minminute := 59, [46].log_data[41].maxminute := 7, [46].log_data[41].valid := 1, [46].log_data[42].min := 2.2917604, [46].log_data[42].max := 2.297178, [46].log_data[42].total := 8261.49, [46].log_data[42].time := 3600.0, [46].log_data[42].minminute := 59, [46].log_data[42].maxminute := 55, [46].log_data[42].valid := 1, [46].log_data[43].min := -0.27999878, [46].log_data[43].max := -0.26000214, [46].log_data[43].total := -991.33185, [46].log_data[43].time := 3600.0, [46].log_data[43].valid := 1, [46].log_data[44].min := -0.3199997, [46].log_data[44].max := -0.30000305,
        [46].log_data[44].total := -1080.1212, [46].log_data[44].time := 3600.0, [46].log_data[44].minminute := 2, [46].log_data[44].valid := 1, [46].log_data[45].time := 3600.0, [46].log_data[45].valid := 1, [46].log_data[46].time := 3600.0, [46].log_data[46].valid := 1, [46].log_data[47].time := 3600.0, [46].log_data[47].valid := 1, [46].log_data[48].min := 6.6852064, [46].log_data[48].max := 6.9536934, [46].log_data[48].total := 24401.06, [46].log_data[48].time := 3600.0, [46].log_data[48].minminute := 59, [46].log_data[48].maxminute := 47, [46].log_data[48].valid := 1, [46].log_data[49].min := 7.194046, [46].log_data[49].max := 9.652006, [46].log_data[49].total := 33094.8, [46].log_data[49].time := 3600.0, [46].log_data[49].minminute := 59, [46].log_data[49].maxminute := 22, [46].log_data[49].valid := 1, [46].log_data[50].min := 1.9992077, [46].log_data[50].max := 2.1517262, [46].log_data[50].total := 7445.122, [46].log_data[50].time := 3600.0, [46].log_data[50].minminute := 23, [46].log_data[50].maxminute := 42, [46].log_data[50].valid := 1, [46].log_data[51].time := 3600.0, [46].log_data[51].valid := 1, [46].log_data[52].min := -4.220001, [46].log_data[52].max := 0.11999512, [46].log_data[52].total := -6917.146, [46].log_data[52].time := 3600.0, [46].log_data[52].minminute := 43, [46].log_data[52].maxminute := 1, [46].log_data[52].valid := 1, [46].log_data[53].min := -3.9399948, [46].log_data[53].max := 0.27999878, [46].log_data[53].total := -6335.2056, [46].log_data[53].time := 3600.0, [46].log_data[53].minminute := 43, [46].log_data[53].maxminute := 18, [46].log_data[53].valid := 1, [46].log_data[54].max := 0.531, [46].log_data[54].total := 835.0584, [46].log_data[54].time := 3600.0, [46].log_data[54].minminute := 1, [46].log_data[54].maxminute := 53, [46].log_data[54].valid := 1, [46].log_data[55].max := 0.5205, [46].log_data[55].total := 813.602, [46].log_data[55].time := 3600.0, [46].log_data[55].minminute := 6, [46].log_data[55].maxminute := 43, [46].log_data[55].valid := 1, [46].log_data[56].min := 0.16028486,
        [46].log_data[56].max := 0.1607167, [46].log_data[56].total := 577.56805, [46].log_data[56].time := 3600.0, [46].log_data[56].minminute := 2, [46].log_data[56].maxminute := 55, [46].log_data[56].valid := 1, [46].log_data[57].min := 0.2814752, [46].log_data[57].max := 0.28190702, [46].log_data[57].total := 1013.8821, [46].log_data[57].time := 3600.0, [46].log_data[57].minminute := 1, [46].log_data[57].maxminute := 37, [46].log_data[57].valid := 1, [46].log_data[58].time := 3600.0, [46].log_data[58].valid := 1, [46].log_data[59].time := 3600.0, [46].log_data[59].valid := 1, [46].log_data[60].valid := 1, [46].log_data[61].valid := 1, [46].log_data[62].valid := 1, [46].log_data[63].valid := 1, [46].log_data[64].valid := 1, [46].log_data[65].valid := 1, [46].log_data[66].valid := 1, [46].log_data[67].valid := 1, [46].log_data[68].valid := 1, [46].log_data[69].valid := 1, [46].log_data[70].valid := 1, [46].log_data[71].valid := 1, [46].log_data[72].valid := 1, [46].log_data[73].valid := 1, [46].log_data[74].valid := 1, [46].log_data[75].valid := 1, [46].log_data[76].valid := 1, [46].log_data[77].valid := 1, [46].log_data[78].valid := 1, [46].log_data[79].valid := 1, [46].log_data[80].valid := 1, [46].log_data[81].valid := 1, [46].log_data[82].valid := 1, [46].log_data[83].valid := 1, [46].log_data[84].valid := 1, [46].log_data[85].valid := 1, [46].log_data[86].valid := 1, [46].log_data[87].valid := 1, [46].log_data[88].valid := 1, [46].log_data[89].valid := 1, [46].log_data[90].valid := 1, [46].log_data[91].valid := 1, [46].log_data[92].valid := 1, [46].log_data[93].valid := 1, [46].log_data[94].valid := 1, [46].log_data[95].valid := 1, [46].log_data[96].valid := 1, [46].log_data[97].valid := 1, [46].log_data[98].valid := 1, [46].log_data[99].valid := 1, [46].log_data[100].valid := 1, [46].log_data[101].valid := 1, [46].log_data[102].valid := 1,
        [46].log_data[103].valid := 1, [46].log_data[104].valid := 1, [46].log_data[105].valid := 1, [46].log_data[106].valid := 1, [46].log_data[107].valid := 1, [46].log_data[108].valid := 1, [46].log_data[109].valid := 1, [46].log_data[110].valid := 1, [46].log_data[111].valid := 1, [46].log_data[112].valid := 1, [46].log_data[113].valid := 1, [46].log_data[114].valid := 1, [46].log_data[115].valid := 1, [46].log_data[116].valid := 1, [46].log_data[117].valid := 1, [46].log_data[118].valid := 1, [46].log_data[119].valid := 1, [46].log_data[120].valid := 1, [46].log_data[121].valid := 1, [46].log_data[122].valid := 1, [46].log_data[123].valid := 1, [46].log_data[124].valid := 1, [46].time.Year := 2023, [46].time.Month := 1, [46].time.Day := 15, [46].time.Hour := 1, [46].time.Minute := 59, [46].time.Second := 59, [47].log_data[0].min := 1.0, [47].log_data[0].max := 1.0, [47].log_data[0].total := 3600.0, [47].log_data[0].time := 3600.0, [47].log_data[0].valid := 1, [47].log_data[1].time := 3600.0, [47].log_data[1].valid := 1, [47].log_data[2].time := 3600.0, [47].log_data[2].valid := 1, [47].log_data[3].time := 3600.0, [47].log_data[3].valid := 1, [47].log_data[4].time := 3600.0, [47].log_data[4].valid := 1, [47].log_data[5].time := 3600.0, [47].log_data[5].valid := 1, [47].log_data[6].time := 3600.0, [47].log_data[6].valid := 1, [47].log_data[7].time := 3600.0, [47].log_data[7].valid := 1, [47].log_data[8].min := 1.0, [47].log_data[8].max := 1.0, [47].log_data[8].total := 3600.0, [47].log_data[8].time := 3600.0, [47].log_data[8].valid := 1, [47].log_data[9].min := 1.0, [47].log_data[9].max := 1.0, [47].log_data[9].total := 3600.0, [47].log_data[9].time := 3600.0, [47].log_data[9].valid := 1, [47].log_data[10].min := 1.0, [47].log_data[10].max := 1.0, [47].log_data[10].total := 3600.0,
        [47].log_data[10].time := 3600.0, [47].log_data[10].valid := 1, [47].log_data[11].time := 3600.0, [47].log_data[11].valid := 1, [47].log_data[12].min := 1.0, [47].log_data[12].max := 1.0, [47].log_data[12].total := 3600.0, [47].log_data[12].time := 3600.0, [47].log_data[12].valid := 1, [47].log_data[13].min := 1.0, [47].log_data[13].max := 1.0, [47].log_data[13].total := 3600.0, [47].log_data[13].time := 3600.0, [47].log_data[13].valid := 1, [47].log_data[14].time := 3600.0, [47].log_data[14].valid := 1, [47].log_data[15].time := 3600.0, [47].log_data[15].valid := 1, [47].log_data[16].time := 3600.0, [47].log_data[16].valid := 1, [47].log_data[17].min := 1.0, [47].log_data[17].max := 1.0, [47].log_data[17].total := 3600.0, [47].log_data[17].time := 3600.0, [47].log_data[17].valid := 1, [47].log_data[18].time := 3600.0, [47].log_data[18].valid := 1, [47].log_data[19].time := 3600.0, [47].log_data[19].valid := 1, [47].log_data[20].time := 3600.0, [47].log_data[20].valid := 1, [47].log_data[21].min := 1.0, [47].log_data[21].max := 1.0, [47].log_data[21].total := 3600.0, [47].log_data[21].time := 3600.0, [47].log_data[21].valid := 1, [47].log_data[22].time := 3600.0, [47].log_data[22].valid := 1, [47].log_data[23].time := 3600.0, [47].log_data[23].valid := 1, [47].log_data[24].time := 3600.0, [47].log_data[24].valid := 1, [47].log_data[25].time := 3600.0, [47].log_data[25].valid := 1, [47].log_data[26].time := 3600.0, [47].log_data[26].valid := 1, [47].log_data[27].time := 3600.0, [47].log_data[27].valid := 1, [47].log_data[28].time := 3600.0, [47].log_data[28].valid := 1, [47].log_data[29].min := 1.0, [47].log_data[29].max := 1.0, [47].log_data[29].total := 3600.0, [47].log_data[29].time := 3600.0, [47].log_data[29].valid := 1, [47].log_data[30].min := 1.0, [47].log_data[30].max := 1.0, [47].log_data[30].total := 3600.0, [47].log_data[30].time := 3600.0, [47].log_data[30].valid := 1,
        [47].log_data[31].max := 1.0, [47].log_data[31].total := 1440.7471, [47].log_data[31].time := 3600.0, [47].log_data[31].minminute := 2, [47].log_data[31].valid := 1, [47].log_data[32].max := 1.0, [47].log_data[32].total := 1629.7471, [47].log_data[32].time := 3600.0, [47].log_data[32].maxminute := 4, [47].log_data[32].valid := 1, [47].log_data[33].time := 3600.0, [47].log_data[33].valid := 1, [47].log_data[34].time := 3600.0, [47].log_data[34].valid := 1, [47].log_data[35].max := 1.0, [47].log_data[35].total := 1588.249, [47].log_data[35].time := 3600.0, [47].log_data[35].minminute := 8, [47].log_data[35].valid := 1, [47].log_data[36].max := 1.0, [47].log_data[36].total := 1570.2471, [47].log_data[36].time := 3600.0, [47].log_data[36].maxminute := 9, [47].log_data[36].valid := 1, [47].log_data[37].time := 3600.0, [47].log_data[37].valid := 1, [47].log_data[38].time := 3600.0, [47].log_data[38].valid := 1, [47].log_data[39].min := 1.004717, [47].log_data[39].max := 1.016259, [47].log_data[39].total := 3639.2437, [47].log_data[39].time := 3600.0, [47].log_data[39].minminute := 54, [47].log_data[39].maxminute := 51, [47].log_data[39].valid := 1, [47].log_data[40].min := 7.5643167, [47].log_data[40].max := 7.604989, [47].log_data[40].total := 27305.639, [47].log_data[40].time := 3600.0, [47].log_data[40].minminute := 12, [47].log_data[40].maxminute := 53, [47].log_data[40].valid := 1, [47].log_data[41].min := 0.026662353, [47].log_data[41].max := 0.037261963, [47].log_data[41].total := 116.19068, [47].log_data[41].time := 3600.0, [47].log_data[41].minminute := 12, [47].log_data[41].maxminute := 36, [47].log_data[41].valid := 1, [47].log_data[42].min := 2.2921138, [47].log_data[42].max := 2.2969427, [47].log_data[42].total := 8261.336, [47].log_data[42].time := 3600.0, [47].log_data[42].minminute := 55, [47].log_data[42].maxminute := 20, [47].log_data[42].valid := 1, [47].log_data[43].min := -0.27999878, [47].log_data[43].max := -0.26000214, [47].log_data[43].total := -969.54913, [47].log_data[43].time := 3600.0,
        [47].log_data[43].valid := 1, [47].log_data[44].min := -0.30000305, [47].log_data[44].max := -0.30000305, [47].log_data[44].total := -1080.0911, [47].log_data[44].time := 3600.0, [47].log_data[44].valid := 1, [47].log_data[45].time := 3600.0, [47].log_data[45].valid := 1, [47].log_data[46].time := 3600.0, [47].log_data[46].valid := 1, [47].log_data[47].time := 3600.0, [47].log_data[47].valid := 1, [47].log_data[48].min := 6.58655, [47].log_data[48].max := 6.7899075, [47].log_data[48].total := 24191.084, [47].log_data[48].time := 3600.0, [47].log_data[48].minminute := 13, [47].log_data[48].maxminute := 26, [47].log_data[48].valid := 1, [47].log_data[49].min := 6.9404373, [47].log_data[49].max := 9.624525, [47].log_data[49].total := 30718.79, [47].log_data[49].time := 3600.0, [47].log_data[49].minminute := 5, [47].log_data[49].maxminute := 57, [47].log_data[49].valid := 1, [47].log_data[50].min := 2.0139296, [47].log_data[50].max := 2.103085, [47].log_data[50].total := 7412.539, [47].log_data[50].time := 3600.0, [47].log_data[50].minminute := 58, [47].log_data[50].valid := 1, [47].log_data[51].time := 3600.0, [47].log_data[51].valid := 1, [47].log_data[52].min := -2.840004, [47].log_data[52].max := 0.11999512, [47].log_data[52].total := -7617.796, [47].log_data[52].time := 3600.0, [47].log_data[52].minminute := 56, [47].log_data[52].maxminute := 2, [47].log_data[52].valid := 1, [47].log_data[53].min := -2.4800034, [47].log_data[53].max := 0.2400055, [47].log_data[53].total := -7193.252, [47].log_data[53].time := 3600.0, [47].log_data[53].minminute := 1, [47].log_data[53].maxminute := 9, [47].log_data[53].valid := 1, [47].log_data[54].max := 0.52, [47].log_data[54].total := 1217.0312, [47].log_data[54].time := 3600.0, [47].log_data[54].minminute := 2, [47].log_data[54].maxminute := 56, [47].log_data[54].valid := 1, [47].log_data[55].max := 0.5175, [47].log_data[55].total := 1253.9572, [47].log_data[55].time := 3600.0, [47].log_data[55].minminute := 8, [47].log_data[55].maxminute := 41, [47].log_data[55].valid := 1,
        [47].log_data[56].min := 0.16020635, [47].log_data[56].max := 0.1607167, [47].log_data[56].total := 577.59186, [47].log_data[56].time := 3600.0, [47].log_data[56].minminute := 10, [47].log_data[56].maxminute := 4, [47].log_data[56].valid := 1, [47].log_data[57].min := 0.2798263, [47].log_data[57].max := 0.28186777, [47].log_data[57].total := 1009.4659, [47].log_data[57].time := 3600.0, [47].log_data[57].minminute := 31, [47].log_data[57].valid := 1, [47].log_data[58].time := 3600.0, [47].log_data[58].valid := 1, [47].log_data[59].time := 3600.0, [47].log_data[59].valid := 1, [47].log_data[60].valid := 1, [47].log_data[61].valid := 1, [47].log_data[62].valid := 1, [47].log_data[63].valid := 1, [47].log_data[64].valid := 1, [47].log_data[65].valid := 1, [47].log_data[66].valid := 1, [47].log_data[67].valid := 1, [47].log_data[68].valid := 1, [47].log_data[69].valid := 1, [47].log_data[70].valid := 1, [47].log_data[71].valid := 1, [47].log_data[72].valid := 1, [47].log_data[73].valid := 1, [47].log_data[74].valid := 1, [47].log_data[75].valid := 1, [47].log_data[76].valid := 1, [47].log_data[77].valid := 1, [47].log_data[78].valid := 1, [47].log_data[79].valid := 1, [47].log_data[80].valid := 1, [47].log_data[81].valid := 1, [47].log_data[82].valid := 1, [47].log_data[83].valid := 1, [47].log_data[84].valid := 1, [47].log_data[85].valid := 1, [47].log_data[86].valid := 1, [47].log_data[87].valid := 1, [47].log_data[88].valid := 1, [47].log_data[89].valid := 1, [47].log_data[90].valid := 1, [47].log_data[91].valid := 1, [47].log_data[92].valid := 1, [47].log_data[93].valid := 1, [47].log_data[94].valid := 1, [47].log_data[95].valid := 1, [47].log_data[96].valid := 1, [47].log_data[97].valid := 1, [47].log_data[98].valid := 1, [47].log_data[99].valid := 1, [47].log_data[100].valid := 1, [47].log_data[101].valid := 1, [47].log_data[102].valid := 1,
        [47].log_data[103].valid := 1, [47].log_data[104].valid := 1, [47].log_data[105].valid := 1, [47].log_data[106].valid := 1, [47].log_data[107].valid := 1, [47].log_data[108].valid := 1, [47].log_data[109].valid := 1, [47].log_data[110].valid := 1, [47].log_data[111].valid := 1, [47].log_data[112].valid := 1, [47].log_data[113].valid := 1, [47].log_data[114].valid := 1, [47].log_data[115].valid := 1, [47].log_data[116].valid := 1, [47].log_data[117].valid := 1, [47].log_data[118].valid := 1, [47].log_data[119].valid := 1, [47].log_data[120].valid := 1, [47].log_data[121].valid := 1, [47].log_data[122].valid := 1, [47].log_data[123].valid := 1, [47].log_data[124].valid := 1, [47].time.Year := 2023, [47].time.Month := 1, [47].time.Day := 15, [47].time.Hour := 2, [47].time.Minute := 59, [47].time.Second := 59, [48].log_data[0].min := 1.0, [48].log_data[0].max := 1.0, [48].log_data[0].total := 3600.0, [48].log_data[0].time := 3600.0, [48].log_data[0].valid := 1, [48].log_data[1].time := 3600.0, [48].log_data[1].valid := 1, [48].log_data[2].time := 3600.0, [48].log_data[2].valid := 1, [48].log_data[3].time := 3600.0, [48].log_data[3].valid := 1, [48].log_data[4].time := 3600.0, [48].log_data[4].valid := 1, [48].log_data[5].time := 3600.0, [48].log_data[5].valid := 1, [48].log_data[6].time := 3600.0, [48].log_data[6].valid := 1, [48].log_data[7].time := 3600.0, [48].log_data[7].valid := 1, [48].log_data[8].max := 1.0, [48].log_data[8].total := 704.251, [48].log_data[8].time := 3600.0, [48].log_data[8].minminute := 11, [48].log_data[8].valid := 1, [48].log_data[9].max := 1.0, [48].log_data[9].total := 704.251, [48].log_data[9].time := 3600.0, [48].log_data[9].minminute := 11, [48].log_data[9].valid := 1, [48].log_data[10].min := 1.0, [48].log_data[10].max := 1.0, [48].log_data[10].total := 3600.0,
        [48].log_data[10].time := 3600.0, [48].log_data[10].valid := 1, [48].log_data[11].time := 3600.0, [48].log_data[11].valid := 1, [48].log_data[12].min := 1.0, [48].log_data[12].max := 1.0, [48].log_data[12].total := 3600.0, [48].log_data[12].time := 3600.0, [48].log_data[12].valid := 1, [48].log_data[13].min := 1.0, [48].log_data[13].max := 1.0, [48].log_data[13].total := 3600.0, [48].log_data[13].time := 3600.0, [48].log_data[13].valid := 1, [48].log_data[14].time := 3600.0, [48].log_data[14].valid := 1, [48].log_data[15].time := 3600.0, [48].log_data[15].valid := 1, [48].log_data[16].time := 3600.0, [48].log_data[16].valid := 1, [48].log_data[17].min := 1.0, [48].log_data[17].max := 1.0, [48].log_data[17].total := 3600.0, [48].log_data[17].time := 3600.0, [48].log_data[17].valid := 1, [48].log_data[18].time := 3600.0, [48].log_data[18].valid := 1, [48].log_data[19].time := 3600.0, [48].log_data[19].valid := 1, [48].log_data[20].time := 3600.0, [48].log_data[20].valid := 1, [48].log_data[21].min := 1.0, [48].log_data[21].max := 1.0, [48].log_data[21].total := 3600.0, [48].log_data[21].time := 3600.0, [48].log_data[21].valid := 1, [48].log_data[22].time := 3600.0, [48].log_data[22].valid := 1, [48].log_data[23].time := 3600.0, [48].log_data[23].valid := 1, [48].log_data[24].time := 3600.0, [48].log_data[24].valid := 1, [48].log_data[25].time := 3600.0, [48].log_data[25].valid := 1, [48].log_data[26].time := 3600.0, [48].log_data[26].valid := 1, [48].log_data[27].time := 3600.0, [48].log_data[27].valid := 1, [48].log_data[28].time := 3600.0, [48].log_data[28].valid := 1, [48].log_data[29].min := 1.0, [48].log_data[29].max := 1.0, [48].log_data[29].total := 3600.0, [48].log_data[29].time := 3600.0, [48].log_data[29].valid := 1, [48].log_data[30].min := 1.0, [48].log_data[30].max := 1.0, [48].log_data[30].total := 3600.0, [48].log_data[30].time := 3600.0, [48].log_data[30].valid := 1,
        [48].log_data[31].max := 1.0, [48].log_data[31].total := 344.0, [48].log_data[31].time := 3600.0, [48].log_data[31].minminute := 5, [48].log_data[31].valid := 1, [48].log_data[32].max := 1.0, [48].log_data[32].total := 275.749, [48].log_data[32].time := 3600.0, [48].log_data[32].maxminute := 7, [48].log_data[32].valid := 1, [48].log_data[33].time := 3600.0, [48].log_data[33].valid := 1, [48].log_data[34].time := 3600.0, [48].log_data[34].valid := 1, [48].log_data[35].max := 1.0, [48].log_data[35].total := 543.0, [48].log_data[35].time := 3600.0, [48].log_data[35].maxminute := 2, [48].log_data[35].valid := 1, [48].log_data[36].max := 1.0, [48].log_data[36].total := 59.5, [48].log_data[36].time := 3600.0, [48].log_data[36].valid := 1, [48].log_data[37].time := 3600.0, [48].log_data[37].valid := 1, [48].log_data[38].time := 3600.0, [48].log_data[38].valid := 1, [48].log_data[39].min := 1.004717, [48].log_data[39].max := 1.0167301, [48].log_data[39].total := 3640.3179, [48].log_data[39].time := 3600.0, [48].log_data[39].minminute := 16, [48].log_data[39].maxminute := 44, [48].log_data[39].valid := 1, [48].log_data[40].min := 7.574485, [48].log_data[40].max := 7.5961943, [48].log_data[40].total := 27309.12, [48].log_data[40].time := 3600.0, [48].log_data[40].minminute := 53, [48].log_data[40].maxminute := 56, [48].log_data[40].valid := 1, [48].log_data[41].min := 0.02273633, [48].log_data[41].max := 0.042169187, [48].log_data[41].total := 104.674835, [48].log_data[41].time := 3600.0, [48].log_data[41].minminute := 11, [48].log_data[41].maxminute := 59, [48].log_data[41].valid := 1, [48].log_data[42].min := 2.2923493, [48].log_data[42].max := 2.2970603, [48].log_data[42].total := 8261.127, [48].log_data[42].time := 3600.0, [48].log_data[42].minminute := 1, [48].log_data[42].maxminute := 1, [48].log_data[42].valid := 1, [48].log_data[43].min := -0.27999878, [48].log_data[43].max := -0.26000214, [48].log_data[43].total := -942.03436, [48].log_data[43].time := 3600.0, [48].log_data[43].valid := 1,
        [48].log_data[44].min := -0.30000305, [48].log_data[44].max := -0.27999878, [48].log_data[44].total := -1077.9817, [48].log_data[44].time := 3600.0, [48].log_data[44].maxminute := 28, [48].log_data[44].valid := 1, [48].log_data[45].time := 3600.0, [48].log_data[45].valid := 1, [48].log_data[46].time := 3600.0, [48].log_data[46].valid := 1, [48].log_data[47].time := 3600.0, [48].log_data[47].valid := 1, [48].log_data[48].min := 6.747862, [48].log_data[48].max := 6.764351, [48].log_data[48].total := 24317.865, [48].log_data[48].time := 3600.0, [48].log_data[48].minminute := 18, [48].log_data[48].maxminute := 59, [48].log_data[48].valid := 1, [48].log_data[49].min := 9.600775, [48].log_data[49].max := 9.673206, [48].log_data[49].total := 34703.72, [48].log_data[49].time := 3600.0, [48].log_data[49].maxminute := 53, [48].log_data[49].valid := 1, [48].log_data[50].min := 1.9992077, [48].log_data[50].max := 2.1113296, [48].log_data[50].total := 7501.705, [48].log_data[50].time := 3600.0, [48].log_data[50].minminute := 11, [48].log_data[50].maxminute := 53, [48].log_data[50].valid := 1, [48].log_data[51].time := 3600.0, [48].log_data[51].valid := 1, [48].log_data[52].min := -2.9400024, [48].log_data[52].max := 0.11999512, [48].log_data[52].total := -5664.5757, [48].log_data[52].time := 3600.0, [48].log_data[52].minminute := 7, [48].log_data[52].maxminute := 5, [48].log_data[52].valid := 1, [48].log_data[53].min := -2.4600067, [48].log_data[53].max := 0.22000122, [48].log_data[53].total := -5111.144, [48].log_data[53].time := 3600.0, [48].log_data[53].minminute := 10, [48].log_data[53].maxminute := 2, [48].log_data[53].valid := 1, [48].log_data[54].max := 0.51100004, [48].log_data[54].total := 246.36977, [48].log_data[54].time := 3600.0, [48].log_data[54].minminute := 5, [48].log_data[54].maxminute := 7, [48].log_data[54].valid := 1, [48].log_data[55].max := 0.49899998, [48].log_data[55].total := 239.5904, [48].log_data[55].time := 3600.0, [48].log_data[55].minminute := 1, [48].log_data[55].maxminute := 2, [48].log_data[55].valid := 1,
        [48].log_data[56].min := 0.16024561, [48].log_data[56].max := 0.16075596, [48].log_data[56].total := 577.6412, [48].log_data[56].time := 3600.0, [48].log_data[56].maxminute := 21, [48].log_data[56].valid := 1, [48].log_data[57].min := 0.27986556, [48].log_data[57].max := 0.28033668, [48].log_data[57].total := 1008.21277, [48].log_data[57].time := 3600.0, [48].log_data[57].minminute := 1, [48].log_data[57].maxminute := 45, [48].log_data[57].valid := 1, [48].log_data[58].time := 3600.0, [48].log_data[58].valid := 1, [48].log_data[59].time := 3600.0, [48].log_data[59].valid := 1, [48].log_data[60].valid := 1, [48].log_data[61].valid := 1, [48].log_data[62].valid := 1, [48].log_data[63].valid := 1, [48].log_data[64].valid := 1, [48].log_data[65].valid := 1, [48].log_data[66].valid := 1, [48].log_data[67].valid := 1, [48].log_data[68].valid := 1, [48].log_data[69].valid := 1, [48].log_data[70].valid := 1, [48].log_data[71].valid := 1, [48].log_data[72].valid := 1, [48].log_data[73].valid := 1, [48].log_data[74].valid := 1, [48].log_data[75].valid := 1, [48].log_data[76].valid := 1, [48].log_data[77].valid := 1, [48].log_data[78].valid := 1, [48].log_data[79].valid := 1, [48].log_data[80].valid := 1, [48].log_data[81].valid := 1, [48].log_data[82].valid := 1, [48].log_data[83].valid := 1, [48].log_data[84].valid := 1, [48].log_data[85].valid := 1, [48].log_data[86].valid := 1, [48].log_data[87].valid := 1, [48].log_data[88].valid := 1, [48].log_data[89].valid := 1, [48].log_data[90].valid := 1, [48].log_data[91].valid := 1, [48].log_data[92].valid := 1, [48].log_data[93].valid := 1, [48].log_data[94].valid := 1, [48].log_data[95].valid := 1, [48].log_data[96].valid := 1, [48].log_data[97].valid := 1, [48].log_data[98].valid := 1, [48].log_data[99].valid := 1, [48].log_data[100].valid := 1, [48].log_data[101].valid := 1, [48].log_data[102].valid := 1,
        [48].log_data[103].valid := 1, [48].log_data[104].valid := 1, [48].log_data[105].valid := 1, [48].log_data[106].valid := 1, [48].log_data[107].valid := 1, [48].log_data[108].valid := 1, [48].log_data[109].valid := 1, [48].log_data[110].valid := 1, [48].log_data[111].valid := 1, [48].log_data[112].valid := 1, [48].log_data[113].valid := 1, [48].log_data[114].valid := 1, [48].log_data[115].valid := 1, [48].log_data[116].valid := 1, [48].log_data[117].valid := 1, [48].log_data[118].valid := 1, [48].log_data[119].valid := 1, [48].log_data[120].valid := 1, [48].log_data[121].valid := 1, [48].log_data[122].valid := 1, [48].log_data[123].valid := 1, [48].log_data[124].valid := 1, [48].time.Year := 2023, [48].time.Month := 1, [48].time.Day := 15, [48].time.Hour := 3, [48].time.Minute := 59, [48].time.Second := 59, [49].log_data[0].min := 1.0, [49].log_data[0].max := 1.0, [49].log_data[0].total := 3600.0, [49].log_data[0].time := 3600.0, [49].log_data[0].valid := 1, [49].log_data[1].max := 1.0, [49].log_data[1].total := 523.5, [49].log_data[1].time := 3600.0, [49].log_data[1].maxminute := 18, [49].log_data[1].valid := 1, [49].log_data[2].max := 1.0, [49].log_data[2].total := 520.0, [49].log_data[2].time := 3600.0, [49].log_data[2].maxminute := 19, [49].log_data[2].valid := 1, [49].log_data[3].time := 3600.0, [49].log_data[3].valid := 1, [49].log_data[4].time := 3600.0, [49].log_data[4].valid := 1, [49].log_data[5].max := 1.0, [49].log_data[5].total := 223.0, [49].log_data[5].time := 3600.0, [49].log_data[5].maxminute := 20, [49].log_data[5].valid := 1, [49].log_data[6].time := 3600.0, [49].log_data[6].valid := 1, [49].log_data[7].time := 3600.0, [49].log_data[7].valid := 1, [49].log_data[8].max := 1.0, [49].log_data[8].total := 2294.749, [49].log_data[8].time := 3600.0, [49].log_data[8].maxminute := 21,
        [49].log_data[8].valid := 1, [49].log_data[9].max := 1.0, [49].log_data[9].total := 2291.249, [49].log_data[9].time := 3600.0, [49].log_data[9].maxminute := 21, [49].log_data[9].valid := 1, [49].log_data[10].min := 1.0, [49].log_data[10].max := 1.0, [49].log_data[10].total := 3600.0, [49].log_data[10].time := 3600.0, [49].log_data[10].valid := 1, [49].log_data[11].time := 3600.0, [49].log_data[11].valid := 1, [49].log_data[12].min := 1.0, [49].log_data[12].max := 1.0, [49].log_data[12].total := 3600.0, [49].log_data[12].time := 3600.0, [49].log_data[12].valid := 1, [49].log_data[13].min := 1.0, [49].log_data[13].max := 1.0, [49].log_data[13].total := 3600.0, [49].log_data[13].time := 3600.0, [49].log_data[13].valid := 1, [49].log_data[14].time := 3600.0, [49].log_data[14].valid := 1, [49].log_data[15].time := 3600.0, [49].log_data[15].valid := 1, [49].log_data[16].time := 3600.0, [49].log_data[16].valid := 1, [49].log_data[17].min := 1.0, [49].log_data[17].max := 1.0, [49].log_data[17].total := 3600.0, [49].log_data[17].time := 3600.0, [49].log_data[17].valid := 1, [49].log_data[18].time := 3600.0, [49].log_data[18].valid := 1, [49].log_data[19].time := 3600.0, [49].log_data[19].valid := 1, [49].log_data[20].time := 3600.0, [49].log_data[20].valid := 1, [49].log_data[21].min := 1.0, [49].log_data[21].max := 1.0, [49].log_data[21].total := 3600.0, [49].log_data[21].time := 3600.0, [49].log_data[21].valid := 1, [49].log_data[22].time := 3600.0, [49].log_data[22].valid := 1, [49].log_data[23].time := 3600.0, [49].log_data[23].valid := 1, [49].log_data[24].time := 3600.0, [49].log_data[24].valid := 1, [49].log_data[25].time := 3600.0, [49].log_data[25].valid := 1, [49].log_data[26].time := 3600.0, [49].log_data[26].valid := 1, [49].log_data[27].time := 3600.0, [49].log_data[27].valid := 1, [49].log_data[28].time := 3600.0, [49].log_data[28].valid := 1, [49].log_data[29].min := 1.0,
        [49].log_data[29].max := 1.0, [49].log_data[29].total := 3600.0, [49].log_data[29].time := 3600.0, [49].log_data[29].valid := 1, [49].log_data[30].min := 1.0, [49].log_data[30].max := 1.0, [49].log_data[30].total := 3600.0, [49].log_data[30].time := 3600.0, [49].log_data[30].valid := 1, [49].log_data[31].max := 1.0, [49].log_data[31].total := 848.247, [49].log_data[31].time := 3600.0, [49].log_data[31].maxminute := 21, [49].log_data[31].valid := 1, [49].log_data[32].max := 1.0, [49].log_data[32].total := 1086.498, [49].log_data[32].time := 3600.0, [49].log_data[32].maxminute := 27, [49].log_data[32].valid := 1, [49].log_data[33].time := 3600.0, [49].log_data[33].valid := 1, [49].log_data[34].time := 3600.0, [49].log_data[34].valid := 1, [49].log_data[35].max := 1.0, [49].log_data[35].total := 932.99805, [49].log_data[35].time := 3600.0, [49].log_data[35].maxminute := 32, [49].log_data[35].valid := 1, [49].log_data[36].max := 1.0, [49].log_data[36].total := 1086.749, [49].log_data[36].time := 3600.0, [49].log_data[36].maxminute := 21, [49].log_data[36].valid := 1, [49].log_data[37].max := 7.601906, [49].log_data[37].total := 3432.411, [49].log_data[37].time := 3600.0, [49].log_data[37].maxminute := 20, [49].log_data[37].valid := 1, [49].log_data[38].time := 3600.0, [49].log_data[38].valid := 1, [49].log_data[39].min := 0.997415, [49].log_data[39].max := 1.0212055, [49].log_data[39].total := 3643.6077, [49].log_data[39].time := 3600.0, [49].log_data[39].minminute := 25, [49].log_data[39].maxminute := 20, [49].log_data[39].valid := 1, [49].log_data[40].min := 7.5544233, [49].log_data[40].max := 7.6047144, [49].log_data[40].total := 27304.744, [49].log_data[40].time := 3600.0, [49].log_data[40].minminute := 41, [49].log_data[40].maxminute := 57, [49].log_data[40].valid := 1, [49].log_data[41].min := 0.03785083, [49].log_data[41].max := 0.050413575, [49].log_data[41].total := 160.28616, [49].log_data[41].time := 3600.0, [49].log_data[41].minminute := 53, [49].log_data[41].maxminute := 9,
        [49].log_data[41].valid := 1, [49].log_data[42].min := 2.2922316, [49].log_data[42].max := 2.2970603, [49].log_data[42].total := 8260.977, [49].log_data[42].time := 3600.0, [49].log_data[42].maxminute := 11, [49].log_data[42].valid := 1, [49].log_data[43].min := -0.27999878, [49].log_data[43].max := -0.26000214, [49].log_data[43].total := -940.3038, [49].log_data[43].time := 3600.0, [49].log_data[43].minminute := 5, [49].log_data[43].valid := 1, [49].log_data[44].min := -0.30000305, [49].log_data[44].max := -0.27999878, [49].log_data[44].total := -1074.7941, [49].log_data[44].time := 3600.0, [49].log_data[44].valid := 1, [49].log_data[45].time := 3600.0, [49].log_data[45].valid := 1, [49].log_data[46].time := 3600.0, [49].log_data[46].valid := 1, [49].log_data[47].time := 3600.0, [49].log_data[47].valid := 1, [49].log_data[48].min := 6.58655, [49].log_data[48].max := 6.9649606, [49].log_data[48].total := 24239.434, [49].log_data[48].time := 3600.0, [49].log_data[48].minminute := 51, [49].log_data[48].maxminute := 26, [49].log_data[48].valid := 1, [49].log_data[49].min := 7.0134583, [49].log_data[49].max := 9.675562, [49].log_data[49].total := 30426.174, [49].log_data[49].time := 3600.0, [49].log_data[49].minminute := 44, [49].log_data[49].maxminute := 11, [49].log_data[49].valid := 1, [49].log_data[50].min := 2.0557399, [49].log_data[50].max := 2.1510196, [49].log_data[50].total := 7537.9062, [49].log_data[50].time := 3600.0, [49].log_data[50].minminute := 59, [49].log_data[50].maxminute := 21, [49].log_data[50].valid := 1, [49].log_data[51].time := 3600.0, [49].log_data[51].valid := 1, [49].log_data[52].min := -4.439995, [49].log_data[52].max := 0.11999512, [49].log_data[52].total := -6801.1807, [49].log_data[52].time := 3600.0, [49].log_data[52].minminute := 21, [49].log_data[52].maxminute := 26, [49].log_data[52].valid := 1, [49].log_data[53].min := -3.9399948, [49].log_data[53].max := 0.22000122, [49].log_data[53].total := -6455.151, [49].log_data[53].time := 3600.0, [49].log_data[53].minminute := 22, [49].log_data[53].maxminute := 31,
        [49].log_data[53].valid := 1, [49].log_data[54].max := 0.549, [49].log_data[54].total := 764.3969, [49].log_data[54].time := 3600.0, [49].log_data[54].maxminute := 59, [49].log_data[54].valid := 1, [49].log_data[55].max := 0.5215, [49].log_data[55].total := 800.2935, [49].log_data[55].time := 3600.0, [49].log_data[55].maxminute := 32, [49].log_data[55].valid := 1, [49].log_data[56].min := 0.16024561, [49].log_data[56].max := 0.16067745, [49].log_data[56].total := 577.4652, [49].log_data[56].time := 3600.0, [49].log_data[56].minminute := 45, [49].log_data[56].valid := 1, [49].log_data[57].min := 0.27860934, [49].log_data[57].max := 0.28033668, [49].log_data[57].total := 1007.7554, [49].log_data[57].time := 3600.0, [49].log_data[57].minminute := 59, [49].log_data[57].maxminute := 31, [49].log_data[57].valid := 1, [49].log_data[58].time := 3600.0, [49].log_data[58].valid := 1, [49].log_data[59].time := 3600.0, [49].log_data[59].valid := 1, [49].log_data[60].valid := 1, [49].log_data[61].valid := 1, [49].log_data[62].valid := 1, [49].log_data[63].valid := 1, [49].log_data[64].valid := 1, [49].log_data[65].valid := 1, [49].log_data[66].valid := 1, [49].log_data[67].valid := 1, [49].log_data[68].valid := 1, [49].log_data[69].valid := 1, [49].log_data[70].valid := 1, [49].log_data[71].valid := 1, [49].log_data[72].valid := 1, [49].log_data[73].valid := 1, [49].log_data[74].valid := 1, [49].log_data[75].valid := 1, [49].log_data[76].valid := 1, [49].log_data[77].valid := 1, [49].log_data[78].valid := 1, [49].log_data[79].valid := 1, [49].log_data[80].valid := 1, [49].log_data[81].valid := 1, [49].log_data[82].valid := 1, [49].log_data[83].valid := 1, [49].log_data[84].valid := 1, [49].log_data[85].valid := 1, [49].log_data[86].valid := 1, [49].log_data[87].valid := 1, [49].log_data[88].valid := 1, [49].log_data[89].valid := 1, [49].log_data[90].valid := 1, [49].log_data[91].valid := 1,
        [49].log_data[92].valid := 1, [49].log_data[93].valid := 1, [49].log_data[94].valid := 1, [49].log_data[95].valid := 1, [49].log_data[96].valid := 1, [49].log_data[97].valid := 1, [49].log_data[98].valid := 1, [49].log_data[99].valid := 1, [49].log_data[100].valid := 1, [49].log_data[101].valid := 1, [49].log_data[102].valid := 1, [49].log_data[103].valid := 1, [49].log_data[104].valid := 1, [49].log_data[105].valid := 1, [49].log_data[106].valid := 1, [49].log_data[107].valid := 1, [49].log_data[108].valid := 1, [49].log_data[109].valid := 1, [49].log_data[110].valid := 1, [49].log_data[111].valid := 1, [49].log_data[112].valid := 1, [49].log_data[113].valid := 1, [49].log_data[114].valid := 1, [49].log_data[115].valid := 1, [49].log_data[116].valid := 1, [49].log_data[117].valid := 1, [49].log_data[118].valid := 1, [49].log_data[119].valid := 1, [49].log_data[120].valid := 1, [49].log_data[121].valid := 1, [49].log_data[122].valid := 1, [49].log_data[123].valid := 1, [49].log_data[124].valid := 1, [49].time.Year := 2023, [49].time.Month := 1, [49].time.Day := 15, [49].time.Hour := 4, [49].time.Minute := 59, [49].time.Second := 59, [50].log_data[0].min := 1.0, [50].log_data[0].max := 1.0, [50].log_data[0].total := 3600.0, [50].log_data[0].time := 3600.0, [50].log_data[0].valid := 1, [50].log_data[1].time := 3600.0, [50].log_data[1].valid := 1, [50].log_data[2].time := 3600.0, [50].log_data[2].valid := 1, [50].log_data[3].time := 3600.0, [50].log_data[3].valid := 1, [50].log_data[4].time := 3600.0, [50].log_data[4].valid := 1, [50].log_data[5].time := 3600.0, [50].log_data[5].valid := 1, [50].log_data[6].time := 3600.0, [50].log_data[6].valid := 1, [50].log_data[7].time := 3600.0, [50].log_data[7].valid := 1, [50].log_data[8].max := 1.0, [50].log_data[8].total := 2623.751,
        [50].log_data[8].time := 3600.0, [50].log_data[8].minminute := 43, [50].log_data[8].valid := 1, [50].log_data[9].max := 1.0, [50].log_data[9].total := 2623.751, [50].log_data[9].time := 3600.0, [50].log_data[9].minminute := 43, [50].log_data[9].valid := 1, [50].log_data[10].min := 1.0, [50].log_data[10].max := 1.0, [50].log_data[10].total := 3600.0, [50].log_data[10].time := 3600.0, [50].log_data[10].valid := 1, [50].log_data[11].time := 3600.0, [50].log_data[11].valid := 1, [50].log_data[12].min := 1.0, [50].log_data[12].max := 1.0, [50].log_data[12].total := 3600.0, [50].log_data[12].time := 3600.0, [50].log_data[12].valid := 1, [50].log_data[13].min := 1.0, [50].log_data[13].max := 1.0, [50].log_data[13].total := 3600.0, [50].log_data[13].time := 3600.0, [50].log_data[13].valid := 1, [50].log_data[14].time := 3600.0, [50].log_data[14].valid := 1, [50].log_data[15].time := 3600.0, [50].log_data[15].valid := 1, [50].log_data[16].time := 3600.0, [50].log_data[16].valid := 1, [50].log_data[17].min := 1.0, [50].log_data[17].max := 1.0, [50].log_data[17].total := 3600.0, [50].log_data[17].time := 3600.0, [50].log_data[17].valid := 1, [50].log_data[18].time := 3600.0, [50].log_data[18].valid := 1, [50].log_data[19].time := 3600.0, [50].log_data[19].valid := 1, [50].log_data[20].time := 3600.0, [50].log_data[20].valid := 1, [50].log_data[21].min := 1.0, [50].log_data[21].max := 1.0, [50].log_data[21].total := 3600.0, [50].log_data[21].time := 3600.0, [50].log_data[21].valid := 1, [50].log_data[22].time := 3600.0, [50].log_data[22].valid := 1, [50].log_data[23].time := 3600.0, [50].log_data[23].valid := 1, [50].log_data[24].time := 3600.0, [50].log_data[24].valid := 1, [50].log_data[25].time := 3600.0, [50].log_data[25].valid := 1, [50].log_data[26].time := 3600.0, [50].log_data[26].valid := 1, [50].log_data[27].time := 3600.0, [50].log_data[27].valid := 1, [50].log_data[28].time := 3600.0,
        [50].log_data[28].valid := 1, [50].log_data[29].min := 1.0, [50].log_data[29].max := 1.0, [50].log_data[29].total := 3600.0, [50].log_data[29].time := 3600.0, [50].log_data[29].valid := 1, [50].log_data[30].min := 1.0, [50].log_data[30].max := 1.0, [50].log_data[30].total := 3600.0, [50].log_data[30].time := 3600.0, [50].log_data[30].valid := 1, [50].log_data[31].max := 1.0, [50].log_data[31].total := 1187.749, [50].log_data[31].time := 3600.0, [50].log_data[31].minminute := 8, [50].log_data[31].valid := 1, [50].log_data[32].max := 1.0, [50].log_data[32].total := 1086.749, [50].log_data[32].time := 3600.0, [50].log_data[32].maxminute := 9, [50].log_data[32].valid := 1, [50].log_data[33].time := 3600.0, [50].log_data[33].valid := 1, [50].log_data[34].time := 3600.0, [50].log_data[34].valid := 1, [50].log_data[35].max := 1.0, [50].log_data[35].total := 1187.998, [50].log_data[35].time := 3600.0, [50].log_data[35].minminute := 2, [50].log_data[35].valid := 1, [50].log_data[36].max := 1.0, [50].log_data[36].total := 1086.749, [50].log_data[36].time := 3600.0, [50].log_data[36].maxminute := 4, [50].log_data[36].valid := 1, [50].log_data[37].time := 3600.0, [50].log_data[37].valid := 1, [50].log_data[38].time := 3600.0, [50].log_data[38].valid := 1, [50].log_data[39].min := 1.0068371, [50].log_data[39].max := 1.0189679, [50].log_data[39].total := 3648.2346, [50].log_data[39].time := 3600.0, [50].log_data[39].minminute := 45, [50].log_data[39].maxminute := 24, [50].log_data[39].valid := 1, [50].log_data[40].min := 7.583004, [50].log_data[40].max := 7.5961943, [50].log_data[40].total := 27314.959, [50].log_data[40].time := 3600.0, [50].log_data[40].minminute := 8, [50].log_data[40].maxminute := 2, [50].log_data[40].valid := 1, [50].log_data[41].min := 0.029802978, [50].log_data[41].max := 0.046487793, [50].log_data[41].total := 143.37384, [50].log_data[41].time := 3600.0, [50].log_data[41].minminute := 32, [50].log_data[41].maxminute := 13, [50].log_data[41].valid := 1,
        [50].log_data[42].min := 2.2918782, [50].log_data[42].max := 2.2969427, [50].log_data[42].total := 8260.8545, [50].log_data[42].time := 3600.0, [50].log_data[42].minminute := 12, [50].log_data[42].maxminute := 12, [50].log_data[42].valid := 1, [50].log_data[43].min := -0.27999878, [50].log_data[43].max := -0.26000214, [50].log_data[43].total := -942.2454, [50].log_data[43].time := 3600.0, [50].log_data[43].valid := 1, [50].log_data[44].min := -0.30000305, [50].log_data[44].max := -0.27999878, [50].log_data[44].total := -1079.729, [50].log_data[44].time := 3600.0, [50].log_data[44].maxminute := 15, [50].log_data[44].valid := 1, [50].log_data[45].time := 3600.0, [50].log_data[45].valid := 1, [50].log_data[46].time := 3600.0, [50].log_data[46].valid := 1, [50].log_data[47].time := 3600.0, [50].log_data[47].valid := 1, [50].log_data[48].min := 6.737969, [50].log_data[48].max := 6.778366, [50].log_data[48].total := 24301.143, [50].log_data[48].time := 3600.0, [50].log_data[48].minminute := 46, [50].log_data[48].maxminute := 4, [50].log_data[48].valid := 1, [50].log_data[49].min := 8.390834, [50].log_data[49].max := 9.6804695, [50].log_data[49].total := 33964.652, [50].log_data[49].time := 3600.0, [50].log_data[49].maxminute := 44, [50].log_data[49].valid := 1, [50].log_data[50].min := 1.9989722, [50].log_data[50].max := 2.1032028, [50].log_data[50].total := 7369.926, [50].log_data[50].time := 3600.0, [50].log_data[50].minminute := 43, [50].log_data[50].maxminute := 58, [50].log_data[50].valid := 1, [50].log_data[51].time := 3600.0, [50].log_data[51].valid := 1, [50].log_data[52].min := -2.9400024, [50].log_data[52].max := 0.11999512, [50].log_data[52].total := -6824.491, [50].log_data[52].time := 3600.0, [50].log_data[52].minminute := 31, [50].log_data[52].maxminute := 8, [50].log_data[52].valid := 1, [50].log_data[53].min := -2.4400024, [50].log_data[53].max := 0.22000122, [50].log_data[53].total := -6245.6978, [50].log_data[53].time := 3600.0, [50].log_data[53].minminute := 1, [50].log_data[53].maxminute := 3, [50].log_data[53].valid := 1,
        [50].log_data[54].max := 0.5415, [50].log_data[54].total := 902.836, [50].log_data[54].time := 3600.0, [50].log_data[54].minminute := 8, [50].log_data[54].maxminute := 20, [50].log_data[54].valid := 1, [50].log_data[55].max := 0.52099997, [50].log_data[55].total := 903.00665, [50].log_data[55].time := 3600.0, [50].log_data[55].minminute := 2, [50].log_data[55].maxminute := 14, [50].log_data[55].valid := 1, [50].log_data[56].min := 0.16020635, [50].log_data[56].max := 0.16063818, [50].log_data[56].total := 577.43286, [50].log_data[56].time := 3600.0, [50].log_data[56].minminute := 49, [50].log_data[56].maxminute := 13, [50].log_data[56].valid := 1, [50].log_data[57].min := 0.2785308, [50].log_data[57].max := 0.27896264, [50].log_data[57].total := 1003.35876, [50].log_data[57].time := 3600.0, [50].log_data[57].minminute := 31, [50].log_data[57].maxminute := 16, [50].log_data[57].valid := 1, [50].log_data[58].time := 3600.0, [50].log_data[58].valid := 1, [50].log_data[59].time := 3600.0, [50].log_data[59].valid := 1, [50].log_data[60].valid := 1, [50].log_data[61].valid := 1, [50].log_data[62].valid := 1, [50].log_data[63].valid := 1, [50].log_data[64].valid := 1, [50].log_data[65].valid := 1, [50].log_data[66].valid := 1, [50].log_data[67].valid := 1, [50].log_data[68].valid := 1, [50].log_data[69].valid := 1, [50].log_data[70].valid := 1, [50].log_data[71].valid := 1, [50].log_data[72].valid := 1, [50].log_data[73].valid := 1, [50].log_data[74].valid := 1, [50].log_data[75].valid := 1, [50].log_data[76].valid := 1, [50].log_data[77].valid := 1, [50].log_data[78].valid := 1, [50].log_data[79].valid := 1, [50].log_data[80].valid := 1, [50].log_data[81].valid := 1, [50].log_data[82].valid := 1, [50].log_data[83].valid := 1, [50].log_data[84].valid := 1, [50].log_data[85].valid := 1, [50].log_data[86].valid := 1, [50].log_data[87].valid := 1, [50].log_data[88].valid := 1, [50].log_data[89].valid := 1,
        [50].log_data[90].valid := 1, [50].log_data[91].valid := 1, [50].log_data[92].valid := 1, [50].log_data[93].valid := 1, [50].log_data[94].valid := 1, [50].log_data[95].valid := 1, [50].log_data[96].valid := 1, [50].log_data[97].valid := 1, [50].log_data[98].valid := 1, [50].log_data[99].valid := 1, [50].log_data[100].valid := 1, [50].log_data[101].valid := 1, [50].log_data[102].valid := 1, [50].log_data[103].valid := 1, [50].log_data[104].valid := 1, [50].log_data[105].valid := 1, [50].log_data[106].valid := 1, [50].log_data[107].valid := 1, [50].log_data[108].valid := 1, [50].log_data[109].valid := 1, [50].log_data[110].valid := 1, [50].log_data[111].valid := 1, [50].log_data[112].valid := 1, [50].log_data[113].valid := 1, [50].log_data[114].valid := 1, [50].log_data[115].valid := 1, [50].log_data[116].valid := 1, [50].log_data[117].valid := 1, [50].log_data[118].valid := 1, [50].log_data[119].valid := 1, [50].log_data[120].valid := 1, [50].log_data[121].valid := 1, [50].log_data[122].valid := 1, [50].log_data[123].valid := 1, [50].log_data[124].valid := 1, [50].time.Year := 2023, [50].time.Month := 1, [50].time.Day := 15, [50].time.Hour := 5, [50].time.Minute := 59, [50].time.Second := 59, [51].log_data[0].min := 1.0, [51].log_data[0].max := 1.0, [51].log_data[0].total := 3600.0, [51].log_data[0].time := 3600.0, [51].log_data[0].valid := 1, [51].log_data[1].time := 3600.0, [51].log_data[1].valid := 1, [51].log_data[2].time := 3600.0, [51].log_data[2].valid := 1, [51].log_data[3].time := 3600.0, [51].log_data[3].valid := 1, [51].log_data[4].time := 3600.0, [51].log_data[4].valid := 1, [51].log_data[5].time := 3600.0, [51].log_data[5].valid := 1, [51].log_data[6].time := 3600.0, [51].log_data[6].valid := 1, [51].log_data[7].time := 3600.0, [51].log_data[7].valid := 1,
        [51].log_data[8].time := 3600.0, [51].log_data[8].valid := 1, [51].log_data[9].time := 3600.0, [51].log_data[9].valid := 1, [51].log_data[10].min := 1.0, [51].log_data[10].max := 1.0, [51].log_data[10].total := 3600.0, [51].log_data[10].time := 3600.0, [51].log_data[10].valid := 1, [51].log_data[11].time := 3600.0, [51].log_data[11].valid := 1, [51].log_data[12].min := 1.0, [51].log_data[12].max := 1.0, [51].log_data[12].total := 3600.0, [51].log_data[12].time := 3600.0, [51].log_data[12].valid := 1, [51].log_data[13].min := 1.0, [51].log_data[13].max := 1.0, [51].log_data[13].total := 3600.0, [51].log_data[13].time := 3600.0, [51].log_data[13].valid := 1, [51].log_data[14].time := 3600.0, [51].log_data[14].valid := 1, [51].log_data[15].time := 3600.0, [51].log_data[15].valid := 1, [51].log_data[16].time := 3600.0, [51].log_data[16].valid := 1, [51].log_data[17].min := 1.0, [51].log_data[17].max := 1.0, [51].log_data[17].total := 3600.0, [51].log_data[17].time := 3600.0, [51].log_data[17].valid := 1, [51].log_data[18].time := 3600.0, [51].log_data[18].valid := 1, [51].log_data[19].time := 3600.0, [51].log_data[19].valid := 1, [51].log_data[20].time := 3600.0, [51].log_data[20].valid := 1, [51].log_data[21].min := 1.0, [51].log_data[21].max := 1.0, [51].log_data[21].total := 3600.0, [51].log_data[21].time := 3600.0, [51].log_data[21].valid := 1, [51].log_data[22].time := 3600.0, [51].log_data[22].valid := 1, [51].log_data[23].time := 3600.0, [51].log_data[23].valid := 1, [51].log_data[24].time := 3600.0, [51].log_data[24].valid := 1, [51].log_data[25].time := 3600.0, [51].log_data[25].valid := 1, [51].log_data[26].time := 3600.0, [51].log_data[26].valid := 1, [51].log_data[27].time := 3600.0, [51].log_data[27].valid := 1, [51].log_data[28].time := 3600.0, [51].log_data[28].valid := 1, [51].log_data[29].min := 1.0, [51].log_data[29].max := 1.0, [51].log_data[29].total := 3600.0,
        [51].log_data[29].time := 3600.0, [51].log_data[29].valid := 1, [51].log_data[30].min := 1.0, [51].log_data[30].max := 1.0, [51].log_data[30].total := 3600.0, [51].log_data[30].time := 3600.0, [51].log_data[30].valid := 1, [51].log_data[31].time := 3600.0, [51].log_data[31].valid := 1, [51].log_data[32].time := 3600.0, [51].log_data[32].valid := 1, [51].log_data[33].time := 3600.0, [51].log_data[33].valid := 1, [51].log_data[34].time := 3600.0, [51].log_data[34].valid := 1, [51].log_data[35].time := 3600.0, [51].log_data[35].valid := 1, [51].log_data[36].time := 3600.0, [51].log_data[36].valid := 1, [51].log_data[37].time := 3600.0, [51].log_data[37].valid := 1, [51].log_data[38].time := 3600.0, [51].log_data[38].valid := 1, [51].log_data[39].min := 1.0062482, [51].log_data[39].max := 1.0189679, [51].log_data[39].total := 3647.8647, [51].log_data[39].time := 3600.0, [51].log_data[39].minminute := 10, [51].log_data[39].maxminute := 39, [51].log_data[39].valid := 1, [51].log_data[40].min := 7.5643167, [51].log_data[40].max := 7.5961943, [51].log_data[40].total := 27310.926, [51].log_data[40].time := 3600.0, [51].log_data[40].minminute := 5, [51].log_data[40].maxminute := 12, [51].log_data[40].valid := 1, [51].log_data[41].min := 0.029802978, [51].log_data[41].max := 0.045309816, [51].log_data[41].total := 128.3821, [51].log_data[41].time := 3600.0, [51].log_data[41].minminute := 42, [51].log_data[41].maxminute := 27, [51].log_data[41].valid := 1, [51].log_data[42].min := 2.2921138, [51].log_data[42].max := 2.296707, [51].log_data[42].total := 8260.669, [51].log_data[42].time := 3600.0, [51].log_data[42].minminute := 49, [51].log_data[42].maxminute := 3, [51].log_data[42].valid := 1, [51].log_data[43].min := -0.27999878, [51].log_data[43].max := -0.26000214, [51].log_data[43].total := -936.278, [51].log_data[43].time := 3600.0, [51].log_data[43].valid := 1, [51].log_data[44].min := -0.30000305, [51].log_data[44].max := -0.27999878, [51].log_data[44].total := -1071.7572, [51].log_data[44].time := 3600.0,
        [51].log_data[44].valid := 1, [51].log_data[45].time := 3600.0, [51].log_data[45].valid := 1, [51].log_data[46].time := 3600.0, [51].log_data[46].valid := 1, [51].log_data[47].time := 3600.0, [51].log_data[47].valid := 1, [51].log_data[48].min := 6.740717, [51].log_data[48].max := 6.759954, [51].log_data[48].total := 24300.557, [51].log_data[48].time := 3600.0, [51].log_data[48].maxminute := 58, [51].log_data[48].valid := 1, [51].log_data[49].min := 9.654558, [51].log_data[49].max := 9.727579, [51].log_data[49].total := 34879.324, [51].log_data[49].time := 3600.0, [51].log_data[49].minminute := 1, [51].log_data[49].maxminute := 53, [51].log_data[49].valid := 1, [51].log_data[50].min := 2.0976675, [51].log_data[50].max := 2.1102695, [51].log_data[50].total := 7582.6924, [51].log_data[50].time := 3600.0, [51].log_data[50].maxminute := 56, [51].log_data[50].valid := 1, [51].log_data[51].time := 3600.0, [51].log_data[51].valid := 1, [51].log_data[52].min := -1.5999985, [51].log_data[52].max := -1.4400024, [51].log_data[52].total := -5422.08, [51].log_data[52].time := 3600.0, [51].log_data[52].minminute := 40, [51].log_data[52].valid := 1, [51].log_data[53].min := -1.5400009, [51].log_data[53].max := -1.3600006, [51].log_data[53].total := -5212.97, [51].log_data[53].time := 3600.0, [51].log_data[53].minminute := 58, [51].log_data[53].valid := 1, [51].log_data[54].time := 3600.0, [51].log_data[54].valid := 1, [51].log_data[55].time := 3600.0, [51].log_data[55].valid := 1, [51].log_data[56].min := 0.16024561, [51].log_data[56].max := 0.16067745, [51].log_data[56].total := 577.5329, [51].log_data[56].time := 3600.0, [51].log_data[56].minminute := 22, [51].log_data[56].maxminute := 8, [51].log_data[56].valid := 1, [51].log_data[57].min := 0.27857006, [51].log_data[57].max := 0.2790019, [51].log_data[57].total := 1003.47375, [51].log_data[57].time := 3600.0, [51].log_data[57].minminute := 5, [51].log_data[57].maxminute := 27, [51].log_data[57].valid := 1, [51].log_data[58].time := 3600.0, [51].log_data[58].valid := 1,
        [51].log_data[59].time := 3600.0, [51].log_data[59].valid := 1, [51].log_data[60].valid := 1, [51].log_data[61].valid := 1, [51].log_data[62].valid := 1, [51].log_data[63].valid := 1, [51].log_data[64].valid := 1, [51].log_data[65].valid := 1, [51].log_data[66].valid := 1, [51].log_data[67].valid := 1, [51].log_data[68].valid := 1, [51].log_data[69].valid := 1, [51].log_data[70].valid := 1, [51].log_data[71].valid := 1, [51].log_data[72].valid := 1, [51].log_data[73].valid := 1, [51].log_data[74].valid := 1, [51].log_data[75].valid := 1, [51].log_data[76].valid := 1, [51].log_data[77].valid := 1, [51].log_data[78].valid := 1, [51].log_data[79].valid := 1, [51].log_data[80].valid := 1, [51].log_data[81].valid := 1, [51].log_data[82].valid := 1, [51].log_data[83].valid := 1, [51].log_data[84].valid := 1, [51].log_data[85].valid := 1, [51].log_data[86].valid := 1, [51].log_data[87].valid := 1, [51].log_data[88].valid := 1, [51].log_data[89].valid := 1, [51].log_data[90].valid := 1, [51].log_data[91].valid := 1, [51].log_data[92].valid := 1, [51].log_data[93].valid := 1, [51].log_data[94].valid := 1, [51].log_data[95].valid := 1, [51].log_data[96].valid := 1, [51].log_data[97].valid := 1, [51].log_data[98].valid := 1, [51].log_data[99].valid := 1, [51].log_data[100].valid := 1, [51].log_data[101].valid := 1, [51].log_data[102].valid := 1, [51].log_data[103].valid := 1, [51].log_data[104].valid := 1, [51].log_data[105].valid := 1, [51].log_data[106].valid := 1, [51].log_data[107].valid := 1, [51].log_data[108].valid := 1, [51].log_data[109].valid := 1, [51].log_data[110].valid := 1, [51].log_data[111].valid := 1, [51].log_data[112].valid := 1, [51].log_data[113].valid := 1, [51].log_data[114].valid := 1, [51].log_data[115].valid := 1, [51].log_data[116].valid := 1, [51].log_data[117].valid := 1,
        [51].log_data[118].valid := 1, [51].log_data[119].valid := 1, [51].log_data[120].valid := 1, [51].log_data[121].valid := 1, [51].log_data[122].valid := 1, [51].log_data[123].valid := 1, [51].log_data[124].valid := 1, [51].time.Year := 2023, [51].time.Month := 1, [51].time.Day := 15, [51].time.Hour := 6, [51].time.Minute := 59, [51].time.Second := 59, [52].log_data[0].min := 1.0, [52].log_data[0].max := 1.0, [52].log_data[0].total := 3600.0, [52].log_data[0].time := 3600.0, [52].log_data[0].valid := 1, [52].log_data[1].time := 3600.0, [52].log_data[1].valid := 1, [52].log_data[2].time := 3600.0, [52].log_data[2].valid := 1, [52].log_data[3].time := 3600.0, [52].log_data[3].valid := 1, [52].log_data[4].time := 3600.0, [52].log_data[4].valid := 1, [52].log_data[5].time := 3600.0, [52].log_data[5].valid := 1, [52].log_data[6].time := 3600.0, [52].log_data[6].valid := 1, [52].log_data[7].time := 3600.0, [52].log_data[7].valid := 1, [52].log_data[8].time := 3600.0, [52].log_data[8].valid := 1, [52].log_data[9].time := 3600.0, [52].log_data[9].valid := 1, [52].log_data[10].min := 1.0, [52].log_data[10].max := 1.0, [52].log_data[10].total := 3600.0, [52].log_data[10].time := 3600.0, [52].log_data[10].valid := 1, [52].log_data[11].time := 3600.0, [52].log_data[11].valid := 1, [52].log_data[12].min := 1.0, [52].log_data[12].max := 1.0, [52].log_data[12].total := 3600.0, [52].log_data[12].time := 3600.0, [52].log_data[12].valid := 1, [52].log_data[13].min := 1.0, [52].log_data[13].max := 1.0, [52].log_data[13].total := 3600.0, [52].log_data[13].time := 3600.0, [52].log_data[13].valid := 1, [52].log_data[14].time := 3600.0, [52].log_data[14].valid := 1, [52].log_data[15].time := 3600.0, [52].log_data[15].valid := 1, [52].log_data[16].time := 3600.0, [52].log_data[16].valid := 1, [52].log_data[17].min := 1.0,
        [52].log_data[17].max := 1.0, [52].log_data[17].total := 3600.0, [52].log_data[17].time := 3600.0, [52].log_data[17].valid := 1, [52].log_data[18].time := 3600.0, [52].log_data[18].valid := 1, [52].log_data[19].time := 3600.0, [52].log_data[19].valid := 1, [52].log_data[20].time := 3600.0, [52].log_data[20].valid := 1, [52].log_data[21].min := 1.0, [52].log_data[21].max := 1.0, [52].log_data[21].total := 3600.0, [52].log_data[21].time := 3600.0, [52].log_data[21].valid := 1, [52].log_data[22].time := 3600.0, [52].log_data[22].valid := 1, [52].log_data[23].time := 3600.0, [52].log_data[23].valid := 1, [52].log_data[24].time := 3600.0, [52].log_data[24].valid := 1, [52].log_data[25].time := 3600.0, [52].log_data[25].valid := 1, [52].log_data[26].time := 3600.0, [52].log_data[26].valid := 1, [52].log_data[27].time := 3600.0, [52].log_data[27].valid := 1, [52].log_data[28].time := 3600.0, [52].log_data[28].valid := 1, [52].log_data[29].min := 1.0, [52].log_data[29].max := 1.0, [52].log_data[29].total := 3600.0, [52].log_data[29].time := 3600.0, [52].log_data[29].valid := 1, [52].log_data[30].min := 1.0, [52].log_data[30].max := 1.0, [52].log_data[30].total := 3600.0, [52].log_data[30].time := 3600.0, [52].log_data[30].valid := 1, [52].log_data[31].time := 3600.0, [52].log_data[31].valid := 1, [52].log_data[32].time := 3600.0, [52].log_data[32].valid := 1, [52].log_data[33].time := 3600.0, [52].log_data[33].valid := 1, [52].log_data[34].time := 3600.0, [52].log_data[34].valid := 1, [52].log_data[35].time := 3600.0, [52].log_data[35].valid := 1, [52].log_data[36].time := 3600.0, [52].log_data[36].valid := 1, [52].log_data[37].time := 3600.0, [52].log_data[37].valid := 1, [52].log_data[38].time := 3600.0, [52].log_data[38].valid := 1, [52].log_data[39].min := 1.0058949, [52].log_data[39].max := 1.0188501, [52].log_data[39].total := 3646.081, [52].log_data[39].time := 3600.0, [52].log_data[39].minminute := 56,
        [52].log_data[39].maxminute := 25, [52].log_data[39].valid := 1, [52].log_data[40].min := 7.5442557, [52].log_data[40].max := 7.5989423, [52].log_data[40].total := 27307.988, [52].log_data[40].time := 3600.0, [52].log_data[40].minminute := 55, [52].log_data[40].maxminute := 48, [52].log_data[40].valid := 1, [52].log_data[41].min := 0.027643798, [52].log_data[41].max := 0.052376464, [52].log_data[41].total := 147.42746, [52].log_data[41].time := 3600.0, [52].log_data[41].minminute := 5, [52].log_data[41].maxminute := 35, [52].log_data[41].valid := 1, [52].log_data[42].min := 2.2917604, [52].log_data[42].max := 2.296707, [52].log_data[42].total := 8260.677, [52].log_data[42].time := 3600.0, [52].log_data[42].minminute := 43, [52].log_data[42].maxminute := 58, [52].log_data[42].valid := 1, [52].log_data[43].min := -0.27999878, [52].log_data[43].max := -0.26000214, [52].log_data[43].total := -946.53973, [52].log_data[43].time := 3600.0, [52].log_data[43].minminute := 4, [52].log_data[43].valid := 1, [52].log_data[44].min := -0.30000305, [52].log_data[44].max := -0.27999878, [52].log_data[44].total := -1078.7457, [52].log_data[44].time := 3600.0, [52].log_data[44].valid := 1, [52].log_data[45].time := 3600.0, [52].log_data[45].valid := 1, [52].log_data[46].time := 3600.0, [52].log_data[46].valid := 1, [52].log_data[47].time := 3600.0, [52].log_data[47].valid := 1, [52].log_data[48].min := 6.7563815, [52].log_data[48].max := 6.767099, [52].log_data[48].total := 24343.002, [52].log_data[48].time := 3600.0, [52].log_data[48].maxminute := 51, [52].log_data[48].valid := 1, [52].log_data[49].min := 9.698725, [52].log_data[49].max := 9.757022, [52].log_data[49].total := 35032.43, [52].log_data[49].time := 3600.0, [52].log_data[49].maxminute := 52, [52].log_data[49].valid := 1, [52].log_data[50].min := 2.1024961, [52].log_data[50].max := 2.1115649, [52].log_data[50].total := 7590.4087, [52].log_data[50].time := 3600.0, [52].log_data[50].minminute := 26, [52].log_data[50].maxminute := 55, [52].log_data[50].valid := 1, [52].log_data[51].time := 3600.0,
